LIN {X 0,Y 538.041,Z 253.279,A -85,B 0,C 180,E1 -4113.632,E2 -4113.632} C_VEL
LIN {X 0,Y 538.013,Z 253.279,A -85,B 0,C 180,E1 -4116.121,E2 -4116.121} C_VEL
LIN {X 0,Y 538.043,Z 253.271,A -85,B 0,C 180,E1 -4119.347,E2 -4119.347} C_VEL
LIN {X 0,Y 538.041,Z 253.271,A -85,B 0,C 180,E1 -4122.466,E2 -4122.466} C_VEL
LIN {X 0,Y 538.068,Z 253.272,A -85,B 0,C 180,E1 -4125.629,E2 -4125.629} C_VEL
LIN {X 0,Y 538.081,Z 253.263,A -85,B 0,C 180,E1 -4128.7,E2 -4128.7} C_VEL
LIN {X 0,Y 538.085,Z 253.27,A -85,B 0,C 180,E1 -4131.737,E2 -4131.737} C_VEL
LIN {X 0,Y 538.121,Z 253.267,A -85,B 0,C 180,E1 -4134,E2 -4134} C_VEL
LIN {X 0,Y 538.128,Z 253.259,A -85,B 0,C 180,E1 -4137.003,E2 -4137.003} C_VEL
LIN {X 0,Y 538.174,Z 253.26,A -85,B 0,C 180,E1 -4139.998,E2 -4139.998} C_VEL
LIN {X 0,Y 538.13,Z 253.259,A -85,B 0,C 180,E1 -4142.992,E2 -4142.992} C_VEL
LIN {X 0,Y 538.108,Z 253.267,A -85,B 0,C 180,E1 -4145.995,E2 -4145.995} C_VEL
LIN {X 0,Y 538.055,Z 253.269,A -85,B 0,C 180,E1 -4149.015,E2 -4149.015} C_VEL
LIN {X 0,Y 538.078,Z 253.272,A -85,B 0,C 180,E1 -4152.06,E2 -4152.06} C_VEL
LIN {X 0,Y 538.038,Z 253.27,A -85,B 0,C 180,E1 -4155.141,E2 -4155.141} C_VEL
LIN {X 0,Y 538.017,Z 253.283,A -85,B 0,C 180,E1 -4158.267,E2 -4158.267} C_VEL
LIN {X 0,Y 538.028,Z 253.277,A -85,B 0,C 180,E1 -4160.648,E2 -4160.648} C_VEL
LIN {X 0,Y 537.991,Z 253.279,A -85,B 0,C 180,E1 -4163.885,E2 -4163.885} C_VEL
LIN {X 0,Y 538.029,Z 253.281,A -85,B 0,C 180,E1 -4166.364,E2 -4166.364} C_VEL
LIN {X 0,Y 538.018,Z 253.277,A -85,B 0,C 180,E1 -4168.931,E2 -4168.931} C_VEL
LIN {X 0,Y 537.997,Z 253.277,A -85,B 0,C 180,E1 -4171.885,E2 -4171.885} C_VEL
LIN {X 0,Y 538.008,Z 253.281,A -85,B 0,C 180,E1 -4174.617,E2 -4174.617} C_VEL
LIN {X 0,Y 537.987,Z 253.28,A -85,B 0,C 180,E1 -4177.167,E2 -4177.167} C_VEL
LIN {X 0,Y 538.01,Z 253.276,A -85,B 0,C 180,E1 -4180.241,E2 -4180.241} C_VEL
LIN {X 0,Y 537.37,Z 253.361,A -85,B 0,C 180,E1 -4180.866,E2 -4180.866} C_VEL
LIN {X 0,Y 534.518,Z 253.716,A -85,B 0,C 180,E1 -4181.881,E2 -4181.881} C_VEL
LIN {X 0,Y 532.084,Z 254.023,A -85,B 0,C 180,E1 -4182.698,E2 -4182.698} C_VEL
LIN {X 0,Y 531.029,Z 254.146,A -85,B 0,C 180,E1 -4183.329,E2 -4183.329} C_VEL
LIN {X 0,Y 530.939,Z 254.156,A -85,B 0,C 180,E1 -4183.543,E2 -4183.543} C_VEL
LIN {X 0,Y 530.94,Z 254.163,A -85,B 0,C 180,E1 -4186.503,E2 -4186.503} C_VEL
LIN {X 0,Y 530.982,Z 254.152,A -85,B 0,C 180,E1 -4189.567,E2 -4189.567} C_VEL
LIN {X 0,Y 530.948,Z 254.163,A -85,B 0,C 180,E1 -4192.573,E2 -4192.573} C_VEL
LIN {X 0,Y 530.982,Z 254.156,A -85,B 0,C 180,E1 -4195.31,E2 -4195.31} C_VEL
LIN {X 0,Y 530.884,Z 254.202,A -85,B 0,C 180,E1 -4196.612,E2 -4196.612} C_VEL
LIN {X 0,Y 530.789,Z 266.896,A -85,B 0,C 180,E1 -4199.38,E2 -4199.38} C_VEL
LIN {X 0,Y 530.787,Z 275.719,A -85,B 0,C 180,E1 -4201.314,E2 -4201.314} C_VEL
LIN {X 0,Y 531.967,Z 284.168,A -85,B 0,C 180,E1 -4201.455,E2 -4201.455} C_VEL
LIN {X 0,Y 531.685,Z 351.425,A -85,B 0,C 180,E1 -4202.382,E2 -4202.382} C_VEL
LIN {X 0,Y 531.589,Z 361.171,A -85,B 0,C 180,E1 -4202.624,E2 -4202.624} C_VEL
LIN {X 0,Y 531.484,Z 372.98,A -85,B 0,C 180,E1 -4203.07,E2 -4203.07} C_VEL
LIN {X 0,Y 531.329,Z 382.663,A -85,B 0,C 180,E1 -4203.592,E2 -4203.592} C_VEL
LIN {X 0,Y 531.152,Z 391.309,A -85,B 0,C 180,E1 -4204.186,E2 -4204.186} C_VEL
LIN {X 0,Y 530.989,Z 398.99,A -85,B 0,C 180,E1 -4204.837,E2 -4204.837} C_VEL
LIN {X 0,Y 530.851,Z 406.002,A -85,B 0,C 180,E1 -4205.561,E2 -4205.561} C_VEL
LIN {X 0,Y 530.738,Z 412.812,A -85,B 0,C 180,E1 -4206.42,E2 -4206.42} C_VEL
LIN {X 0,Y 530.635,Z 419.151,A -85,B 0,C 180,E1 -4207.413,E2 -4207.413} C_VEL
LIN {X 0,Y 530.543,Z 423.279,A -85,B 0,C 180,E1 -4208.228,E2 -4208.228} C_VEL
LIN {X 0,Y 530.505,Z 427.975,A -85,B 0,C 180,E1 -4209.448,E2 -4209.448} C_VEL
LIN {X 0,Y 530.483,Z 430.043,A -85,B 0,C 180,E1 -4210.145,E2 -4210.145} C_VEL
LIN {X 0,Y 530.384,Z 432.54,A -85,B 0,C 180,E1 -4211.457,E2 -4211.457} C_VEL
LIN {X 0,Y 530.398,Z 433.506,A -85,B 0,C 180,E1 -4212.545,E2 -4212.545} C_VEL
LIN {X 0,Y 530.42,Z 433.688,A -85,B 0,C 180,E1 -4213.053,E2 -4213.053} C_VEL
LIN {X 0,Y 530.396,Z 433.379,A -85,B 0,C 180,E1 -4213.844,E2 -4213.844} C_VEL
LIN {X 0,Y 530.412,Z 432.535,A -85,B 0,C 180,E1 -4214.633,E2 -4214.633} C_VEL
LIN {X 0,Y 530.456,Z 431.175,A -85,B 0,C 180,E1 -4215.42,E2 -4215.42} C_VEL
LIN {X 0,Y 530.509,Z 428.107,A -85,B 0,C 180,E1 -4216.595,E2 -4216.595} C_VEL
LIN {X 0,Y 530.556,Z 423.719,A -85,B 0,C 180,E1 -4217.764,E2 -4217.764} C_VEL
LIN {X 0,Y 530.654,Z 419.171,A -85,B 0,C 180,E1 -4218.671,E2 -4218.671} C_VEL
LIN {X 0,Y 530.728,Z 412.559,A -85,B 0,C 180,E1 -4219.702,E2 -4219.702} C_VEL
LIN {X 0,Y 530.856,Z 406.455,A -85,B 0,C 180,E1 -4220.475,E2 -4220.475} C_VEL
LIN {X 0,Y 531.014,Z 399.031,A -85,B 0,C 180,E1 -4221.246,E2 -4221.246} C_VEL
LIN {X 0,Y 531.138,Z 391.103,A -85,B 0,C 180,E1 -4221.918,E2 -4221.918} C_VEL
LIN {X 0,Y 531.308,Z 381.979,A -85,B 0,C 180,E1 -4222.54,E2 -4222.54} C_VEL
LIN {X 0,Y 531.46,Z 371.213,A -85,B 0,C 180,E1 -4223.097,E2 -4223.097} C_VEL
LIN {X 0,Y 531.575,Z 360.799,A -85,B 0,C 180,E1 -4223.476,E2 -4223.476} C_VEL
LIN {X 0,Y 531.7,Z 350.946,A -85,B 0,C 180,E1 -4223.716,E2 -4223.716} C_VEL
LIN {X 0,Y 531.779,Z 281.945,A -85,B 0,C 180,E1 -4224.668,E2 -4224.668} C_VEL
LIN {X 0,Y 530.812,Z 275.687,A -85,B 0,C 180,E1 -4224.778,E2 -4224.778} C_VEL
LIN {X 0,Y 530.914,Z 261.115,A -85,B 0,C 180,E1 -4228.104,E2 -4228.104} C_VEL
LIN {X 0,Y 530.937,Z 254.161,A -85,B 0,C 180,E1 -4229.716,E2 -4229.716} C_VEL
LIN {X 0,Y 531.118,Z 254.139,A -85,B 0,C 180,E1 -4230.758,E2 -4230.758} C_VEL
LIN {X 0,Y 531.072,Z 254.145,A -85,B 0,C 180,E1 -4233.034,E2 -4233.034} C_VEL
LIN {X 0,Y 531.04,Z 254.144,A -85,B 0,C 180,E1 -4236.078,E2 -4236.078} C_VEL
LIN {X 0,Y 530.988,Z 254.157,A -85,B 0,C 180,E1 -4239.139,E2 -4239.139} C_VEL
LIN {X 0,Y 531.021,Z 254.15,A -85,B 0,C 180,E1 -4241.677,E2 -4241.677} C_VEL
LIN {X 0,Y 530.991,Z 254.153,A -85,B 0,C 180,E1 -4244.956,E2 -4244.956} C_VEL
LIN {X 0,Y 530.979,Z 254.155,A -85,B 0,C 180,E1 -4247.724,E2 -4247.724} C_VEL
LIN {X 0,Y 530.988,Z 254.15,A -85,B 0,C 180,E1 -4250.129,E2 -4250.129} C_VEL
LIN {X 0,Y 530.907,Z 254.16,A -85,B 0,C 180,E1 -4252.575,E2 -4252.575} C_VEL
LIN {X 0,Y 530.925,Z 254.161,A -85,B 0,C 180,E1 -4255.062,E2 -4255.062} C_VEL
LIN {X 0,Y 530.937,Z 254.164,A -85,B 0,C 180,E1 -4257.6,E2 -4257.6} C_VEL
LIN {X 0,Y 530.926,Z 254.158,A -85,B 0,C 180,E1 -4260.2,E2 -4260.2} C_VEL
LIN {X 0,Y 530.936,Z 254.157,A -85,B 0,C 180,E1 -4262.869,E2 -4262.869} C_VEL
LIN {X 0,Y 530.919,Z 254.167,A -85,B 0,C 180,E1 -4265.623,E2 -4265.623} C_VEL
LIN {X 0,Y 530.933,Z 254.157,A -85,B 0,C 180,E1 -4268.656,E2 -4268.656} C_VEL
LIN {X 0,Y 530.952,Z 254.161,A -85,B 0,C 180,E1 -4271.44,E2 -4271.44} C_VEL
LIN {X 0,Y 530.949,Z 254.155,A -85,B 0,C 180,E1 -4274.551,E2 -4274.551} C_VEL
LIN {X 0,Y 530.96,Z 254.16,A -85,B 0,C 180,E1 -4277.837,E2 -4277.837} C_VEL
LIN {X 0,Y 530.963,Z 254.153,A -85,B 0,C 180,E1 -4280.559,E2 -4280.559} C_VEL
LIN {X 0,Y 530.934,Z 254.162,A -85,B 0,C 180,E1 -4283.444,E2 -4283.444} C_VEL
LIN {X 0,Y 530.939,Z 254.158,A -85,B 0,C 180,E1 -4286.228,E2 -4286.228} C_VEL
LIN {X 0,Y 530.96,Z 254.158,A -85,B 0,C 180,E1 -4289.358,E2 -4289.358} C_VEL
LIN {X 0,Y 530.951,Z 254.161,A -85,B 0,C 180,E1 -4291.546,E2 -4291.546} C_VEL
LIN {X 0,Y 530.963,Z 254.157,A -85,B 0,C 180,E1 -4294.168,E2 -4294.168} C_VEL
LIN {X 0,Y 530.943,Z 254.156,A -85,B 0,C 180,E1 -4296.606,E2 -4296.606} C_VEL
LIN {X 0,Y 530.99,Z 254.151,A -85,B 0,C 180,E1 -4299.065,E2 -4299.065} C_VEL
LIN {X 0,Y 530.964,Z 254.158,A -85,B 0,C 180,E1 -4301.481,E2 -4301.481} C_VEL
LIN {X 0,Y 530.961,Z 254.324,A -85,B 0,C 180,E1 -4303.321,E2 -4303.321} C_VEL
LIN {X 0,Y 530.917,Z 265.036,A -85,B 0,C 180,E1 -4305.828,E2 -4305.828} C_VEL
LIN {X 0,Y 530.785,Z 275.645,A -85,B 0,C 180,E1 -4308.323,E2 -4308.323} C_VEL
LIN {X 0,Y 531.892,Z 283.251,A -85,B 0,C 180,E1 -4308.465,E2 -4308.465} C_VEL
LIN {X 0,Y 531.64,Z 352.125,A -85,B 0,C 180,E1 -4309.434,E2 -4309.434} C_VEL
LIN {X 0,Y 531.525,Z 363.522,A -85,B 0,C 180,E1 -4309.744,E2 -4309.744} C_VEL
LIN {X 0,Y 531.334,Z 374.684,A -85,B 0,C 180,E1 -4310.198,E2 -4310.198} C_VEL
LIN {X 0,Y 531.216,Z 384.815,A -85,B 0,C 180,E1 -4310.772,E2 -4310.772} C_VEL
LIN {X 0,Y 531.091,Z 393.972,A -85,B 0,C 180,E1 -4311.441,E2 -4311.441} C_VEL
LIN {X 0,Y 530.918,Z 402.344,A -85,B 0,C 180,E1 -4312.205,E2 -4312.205} C_VEL
LIN {X 0,Y 530.758,Z 410.574,A -85,B 0,C 180,E1 -4313.158,E2 -4313.158} C_VEL
LIN {X 0,Y 530.717,Z 417.097,A -85,B 0,C 180,E1 -4314.112,E2 -4314.112} C_VEL
LIN {X 0,Y 530.581,Z 422.263,A -85,B 0,C 180,E1 -4315.063,E2 -4315.063} C_VEL
LIN {X 0,Y 530.56,Z 425.573,A -85,B 0,C 180,E1 -4315.825,E2 -4315.825} C_VEL
LIN {X 0,Y 530.527,Z 429.412,A -85,B 0,C 180,E1 -4316.965,E2 -4316.965} C_VEL
LIN {X 0,Y 530.412,Z 431.261,A -85,B 0,C 180,E1 -4317.724,E2 -4317.724} C_VEL
LIN {X 0,Y 530.363,Z 432.569,A -85,B 0,C 180,E1 -4318.484,E2 -4318.484} C_VEL
LIN {X 0,Y 530.355,Z 433.359,A -85,B 0,C 180,E1 -4319.243,E2 -4319.243} C_VEL
LIN {X 0,Y 530.357,Z 433.615,A -85,B 0,C 180,E1 -4320.002,E2 -4320.002} C_VEL
LIN {X 0,Y 530.357,Z 433.432,A -85,B 0,C 180,E1 -4320.762,E2 -4320.762} C_VEL
LIN {X 0,Y 530.363,Z 432.692,A -85,B 0,C 180,E1 -4321.521,E2 -4321.521} C_VEL
LIN {X 0,Y 530.414,Z 431.453,A -85,B 0,C 180,E1 -4322.28,E2 -4322.28} C_VEL
LIN {X 0,Y 530.549,Z 428.597,A -85,B 0,C 180,E1 -4323.42,E2 -4323.42} C_VEL
LIN {X 0,Y 530.604,Z 424.486,A -85,B 0,C 180,E1 -4324.56,E2 -4324.56} C_VEL
LIN {X 0,Y 530.659,Z 418.8,A -85,B 0,C 180,E1 -4325.703,E2 -4325.703} C_VEL
LIN {X 0,Y 530.729,Z 412.348,A -85,B 0,C 180,E1 -4326.702,E2 -4326.702} C_VEL
LIN {X 0,Y 530.87,Z 404.997,A -85,B 0,C 180,E1 -4327.61,E2 -4327.61} C_VEL
LIN {X 0,Y 531.037,Z 396.186,A -85,B 0,C 180,E1 -4328.469,E2 -4328.469} C_VEL
LIN {X 0,Y 531.245,Z 387.509,A -85,B 0,C 180,E1 -4329.137,E2 -4329.137} C_VEL
LIN {X 0,Y 531.351,Z 378.086,A -85,B 0,C 180,E1 -4329.711,E2 -4329.711} C_VEL
LIN {X 0,Y 531.489,Z 367.857,A -85,B 0,C 180,E1 -4330.189,E2 -4330.189} C_VEL
LIN {X 0,Y 531.58,Z 356.589,A -85,B 0,C 180,E1 -4330.548,E2 -4330.548} C_VEL
LIN {X 0,Y 531.737,Z 343.655,A -85,B 0,C 180,E1 -4330.786,E2 -4330.786} C_VEL
LIN {X 0,Y 531.751,Z 281.777,A -85,B 0,C 180,E1 -4331.649,E2 -4331.649} C_VEL
LIN {X 0,Y 530.789,Z 275.755,A -85,B 0,C 180,E1 -4331.767,E2 -4331.767} C_VEL
LIN {X 0,Y 530.888,Z 265.704,A -85,B 0,C 180,E1 -4334.178,E2 -4334.178} C_VEL
LIN {X 0,Y 531.002,Z 254.155,A -85,B 0,C 180,E1 -4336.782,E2 -4336.782} C_VEL
LIN {X 0,Y 531.033,Z 254.155,A -85,B 0,C 180,E1 -4340.129,E2 -4340.129} C_VEL
LIN {X 0,Y 530.951,Z 254.161,A -85,B 0,C 180,E1 -4342.575,E2 -4342.575} C_VEL
LIN {X 0,Y 530.959,Z 254.156,A -85,B 0,C 180,E1 -4345.062,E2 -4345.062} C_VEL
LIN {X 0,Y 530.973,Z 254.154,A -85,B 0,C 180,E1 -4347.599,E2 -4347.599} C_VEL
LIN {X 0,Y 530.961,Z 254.161,A -85,B 0,C 180,E1 -4350.199,E2 -4350.199} C_VEL
LIN {X 0,Y 530.975,Z 254.156,A -85,B 0,C 180,E1 -4352.868,E2 -4352.868} C_VEL
LIN {X 0,Y 530.956,Z 254.155,A -85,B 0,C 180,E1 -4355.621,E2 -4355.621} C_VEL
LIN {X 0,Y 530.971,Z 254.16,A -85,B 0,C 180,E1 -4358.654,E2 -4358.654} C_VEL
LIN {X 0,Y 530.987,Z 254.151,A -85,B 0,C 180,E1 -4361.438,E2 -4361.438} C_VEL
LIN {X 0,Y 530.98,Z 254.159,A -85,B 0,C 180,E1 -4364.549,E2 -4364.549} C_VEL
LIN {X 0,Y 530.976,Z 254.152,A -85,B 0,C 180,E1 -4367.836,E2 -4367.836} C_VEL
LIN {X 0,Y 530.99,Z 254.158,A -85,B 0,C 180,E1 -4370.557,E2 -4370.557} C_VEL
LIN {X 0,Y 530.957,Z 254.153,A -85,B 0,C 180,E1 -4373.441,E2 -4373.441} C_VEL
LIN {X 0,Y 530.961,Z 254.156,A -85,B 0,C 180,E1 -4376.225,E2 -4376.225} C_VEL
LIN {X 0,Y 530.96,Z 254.161,A -85,B 0,C 180,E1 -4378.921,E2 -4378.921} C_VEL
LIN {X 0,Y 530.978,Z 254.153,A -85,B 0,C 180,E1 -4381.543,E2 -4381.543} C_VEL
LIN {X 0,Y 531.018,Z 254.149,A -85,B 0,C 180,E1 -4384.156,E2 -4384.156} C_VEL
LIN {X 0,Y 531.044,Z 254.342,A -85,B 0,C 180,E1 -4386.814,E2 -4386.814} C_VEL
LIN {X 0,Y 531.791,Z 259.167,A -85,B 0,C 180,E1 -4387.685,E2 -4387.685} C_VEL
LIN {X 0,Y 531.629,Z 273.173,A -85,B 0,C 180,E1 -4390.098,E2 -4390.098} C_VEL
LIN {X 0,Y 531.34,Z 289.579,A -85,B 0,C 180,E1 -4392.884,E2 -4392.884} C_VEL
LIN {X 0,Y 531.07,Z 308.295,A -85,B 0,C 180,E1 -4396.024,E2 -4396.024} C_VEL
LIN {X 0,Y 530.887,Z 321.55,A -85,B 0,C 180,E1 -4398.231,E2 -4398.231} C_VEL
LIN {X 0,Y 531.888,Z 330.701,A -85,B 0,C 180,E1 -4398.389,E2 -4398.389} C_VEL
LIN {X 0,Y 531.659,Z 399.476,A -85,B 0,C 180,E1 -4399.335,E2 -4399.335} C_VEL
LIN {X 0,Y 531.516,Z 409.998,A -85,B 0,C 180,E1 -4399.597,E2 -4399.597} C_VEL
LIN {X 0,Y 531.364,Z 420.758,A -85,B 0,C 180,E1 -4400.003,E2 -4400.003} C_VEL
LIN {X 0,Y 531.221,Z 431.422,A -85,B 0,C 180,E1 -4400.577,E2 -4400.577} C_VEL
LIN {X 0,Y 531.118,Z 439.774,A -85,B 0,C 180,E1 -4401.151,E2 -4401.151} C_VEL
LIN {X 0,Y 530.931,Z 447.675,A -85,B 0,C 180,E1 -4401.819,E2 -4401.819} C_VEL
LIN {X 0,Y 530.786,Z 455.064,A -85,B 0,C 180,E1 -4402.582,E2 -4402.582} C_VEL
LIN {X 0,Y 530.669,Z 462.835,A -85,B 0,C 180,E1 -4403.575,E2 -4403.575} C_VEL
LIN {X 0,Y 530.542,Z 469.414,A -85,B 0,C 180,E1 -4404.679,E2 -4404.679} C_VEL
LIN {X 0,Y 530.544,Z 474.617,A -85,B 0,C 180,E1 -4405.822,E2 -4405.822} C_VEL
LIN {X 0,Y 530.47,Z 478.434,A -85,B 0,C 180,E1 -4406.962,E2 -4406.962} C_VEL
LIN {X 0,Y 530.413,Z 480.189,A -85,B 0,C 180,E1 -4407.722,E2 -4407.722} C_VEL
LIN {X 0,Y 530.36,Z 481.446,A -85,B 0,C 180,E1 -4408.481,E2 -4408.481} C_VEL
LIN {X 0,Y 530.347,Z 482.23,A -85,B 0,C 180,E1 -4409.241,E2 -4409.241} C_VEL
LIN {X 0,Y 530.349,Z 482.526,A -85,B 0,C 180,E1 -4410,E2 -4410} C_VEL
LIN {X 0,Y 530.347,Z 482.228,A -85,B 0,C 180,E1 -4410.759,E2 -4410.759} C_VEL
LIN {X 0,Y 530.36,Z 481.444,A -85,B 0,C 180,E1 -4411.519,E2 -4411.519} C_VEL
LIN {X 0,Y 530.413,Z 480.185,A -85,B 0,C 180,E1 -4412.278,E2 -4412.278} C_VEL
LIN {X 0,Y 530.494,Z 477.269,A -85,B 0,C 180,E1 -4413.418,E2 -4413.418} C_VEL
LIN {X 0,Y 530.544,Z 474.61,A -85,B 0,C 180,E1 -4414.178,E2 -4414.178} C_VEL
LIN {X 0,Y 530.542,Z 469.402,A -85,B 0,C 180,E1 -4415.32,E2 -4415.32} C_VEL
LIN {X 0,Y 530.673,Z 462.787,A -85,B 0,C 180,E1 -4416.429,E2 -4416.429} C_VEL
LIN {X 0,Y 530.786,Z 455.052,A -85,B 0,C 180,E1 -4417.417,E2 -4417.417} C_VEL
LIN {X 0,Y 530.929,Z 447.664,A -85,B 0,C 180,E1 -4418.181,E2 -4418.181} C_VEL
LIN {X 0,Y 531.097,Z 439.756,A -85,B 0,C 180,E1 -4418.849,E2 -4418.849} C_VEL
LIN {X 0,Y 531.221,Z 431.401,A -85,B 0,C 180,E1 -4419.423,E2 -4419.423} C_VEL
LIN {X 0,Y 531.364,Z 420.737,A -85,B 0,C 180,E1 -4419.997,E2 -4419.997} C_VEL
LIN {X 0,Y 531.525,Z 409.145,A -85,B 0,C 180,E1 -4420.427,E2 -4420.427} C_VEL
LIN {X 0,Y 531.652,Z 399.452,A -85,B 0,C 180,E1 -4420.665,E2 -4420.665} C_VEL
LIN {X 0,Y 531.882,Z 330.638,A -85,B 0,C 180,E1 -4421.612,E2 -4421.612} C_VEL
LIN {X 0,Y 530.891,Z 321.475,A -85,B 0,C 180,E1 -4421.77,E2 -4421.77} C_VEL
LIN {X 0,Y 531.107,Z 302.114,A -85,B 0,C 180,E1 -4424.985,E2 -4424.985} C_VEL
LIN {X 0,Y 531.411,Z 283.707,A -85,B 0,C 180,E1 -4428.067,E2 -4428.067} C_VEL
LIN {X 0,Y 531.701,Z 265.728,A -85,B 0,C 180,E1 -4431.112,E2 -4431.112} C_VEL
LIN {X 0,Y 531.732,Z 258.797,A -85,B 0,C 180,E1 -4432.3,E2 -4432.3} C_VEL
LIN {X 0,Y 531.015,Z 254.156,A -85,B 0,C 180,E1 -4433.136,E2 -4433.136} C_VEL
LIN {X 0,Y 531.016,Z 254.149,A -85,B 0,C 180,E1 -4435.897,E2 -4435.897} C_VEL
LIN {X 0,Y 530.976,Z 254.153,A -85,B 0,C 180,E1 -4438.457,E2 -4438.457} C_VEL
LIN {X 0,Y 530.958,Z 254.16,A -85,B 0,C 180,E1 -4441.079,E2 -4441.079} C_VEL
LIN {X 0,Y 530.96,Z 254.158,A -85,B 0,C 180,E1 -4443.775,E2 -4443.775} C_VEL
LIN {X 0,Y 530.959,Z 254.152,A -85,B 0,C 180,E1 -4446.558,E2 -4446.558} C_VEL
LIN {X 0,Y 530.989,Z 254.159,A -85,B 0,C 180,E1 -4449.443,E2 -4449.443} C_VEL
LIN {X 0,Y 530.979,Z 254.151,A -85,B 0,C 180,E1 -4452.456,E2 -4452.456} C_VEL
LIN {X 0,Y 530.981,Z 254.159,A -85,B 0,C 180,E1 -4455.622,E2 -4455.622} C_VEL
LIN {X 0,Y 530.999,Z 254.148,A -85,B 0,C 180,E1 -4458.563,E2 -4458.563} C_VEL
LIN {X 0,Y 530.961,Z 254.16,A -85,B 0,C 180,E1 -4461.528,E2 -4461.528} C_VEL
LIN {X 0,Y 530.959,Z 254.152,A -85,B 0,C 180,E1 -4464.379,E2 -4464.379} C_VEL
LIN {X 0,Y 530.972,Z 254.154,A -85,B 0,C 180,E1 -4467.132,E2 -4467.132} C_VEL
LIN {X 0,Y 530.96,Z 254.161,A -85,B 0,C 180,E1 -4469.801,E2 -4469.801} C_VEL
LIN {X 0,Y 530.979,Z 254.151,A -85,B 0,C 180,E1 -4472.475,E2 -4472.475} C_VEL
LIN {X 0,Y 530.994,Z 254.149,A -85,B 0,C 180,E1 -4474.94,E2 -4474.94} C_VEL
LIN {X 0,Y 530.977,Z 254.152,A -85,B 0,C 180,E1 -4478.245,E2 -4478.245} C_VEL
LIN {X 0,Y 530.988,Z 254.15,A -85,B 0,C 180,E1 -4480.675,E2 -4480.675} C_VEL
LIN {X 0,Y 530.974,Z 254.15,A -85,B 0,C 180,E1 -4483.069,E2 -4483.069} C_VEL
LIN {X 0,Y 531.024,Z 254.146,A -85,B 0,C 180,E1 -4485.434,E2 -4485.434} C_VEL
LIN {X 0,Y 531.039,Z 254.141,A -85,B 0,C 180,E1 -4488.548,E2 -4488.548} C_VEL
LIN {X 0,Y 531.054,Z 254.144,A -85,B 0,C 180,E1 -4491.627,E2 -4491.627} C_VEL
LIN {X 0,Y 531.119,Z 254.131,A -85,B 0,C 180,E1 -4494.683,E2 -4494.683} C_VEL
LIN {X 0,Y 531.14,Z 254.134,A -85,B 0,C 180,E1 -4497.723,E2 -4497.723} C_VEL
LIN {X 0,Y 531.147,Z 254.129,A -85,B 0,C 180,E1 -4500.756,E2 -4500.756} C_VEL
LIN {X 0,Y 531.098,Z 254.135,A -85,B 0,C 180,E1 -4503.032,E2 -4503.032} C_VEL
LIN {X 0,Y 531.064,Z 254.145,A -85,B 0,C 180,E1 -4506.075,E2 -4506.075} C_VEL
LIN {X 0,Y 531.015,Z 254.145,A -85,B 0,C 180,E1 -4509.136,E2 -4509.136} C_VEL
LIN {X 0,Y 531.035,Z 254.152,A -85,B 0,C 180,E1 -4512.222,E2 -4512.222} C_VEL
LIN {X 0,Y 530.988,Z 254.148,A -85,B 0,C 180,E1 -4515.347,E2 -4515.347} C_VEL
LIN {X 0,Y 530.977,Z 254.157,A -85,B 0,C 180,E1 -4518.518,E2 -4518.518} C_VEL
LIN {X 0,Y 530.989,Z 254.151,A -85,B 0,C 180,E1 -4520.935,E2 -4520.935} C_VEL
LIN {X 0,Y 530.959,Z 254.16,A -85,B 0,C 180,E1 -4524.222,E2 -4524.222} C_VEL
LIN {X 0,Y 530.993,Z 254.154,A -85,B 0,C 180,E1 -4526.741,E2 -4526.741} C_VEL
LIN {X 0,Y 530.968,Z 254.153,A -85,B 0,C 180,E1 -4529.319,E2 -4529.319} C_VEL
LIN {X 0,Y 530.953,Z 254.157,A -85,B 0,C 180,E1 -4532.098,E2 -4532.098} C_VEL
LIN {X 0,Y 530.965,Z 254.155,A -85,B 0,C 180,E1 -4534.85,E2 -4534.85} C_VEL
LIN {X 0,Y 530.946,Z 254.155,A -85,B 0,C 180,E1 -4537.505,E2 -4537.505} C_VEL
LIN {X 0,Y 530.978,Z 254.157,A -85,B 0,C 180,E1 -4540.428,E2 -4540.428} C_VEL
LIN {X 0,Y 530.942,Z 254.156,A -85,B 0,C 180,E1 -4543.492,E2 -4543.492} C_VEL
LIN {X 0,Y 530.939,Z 254.156,A -85,B 0,C 180,E1 -4543.543,E2 -4543.543} C_VEL
LIN {X 0,Y 530.264,Z 254.243,A -85,B 0,C 180,E1 -4544.176,E2 -4544.176} C_VEL
LIN {X 0,Y 527.417,Z 254.604,A -85,B 0,C 180,E1 -4545.205,E2 -4545.205} C_VEL
LIN {X 0,Y 525.015,Z 254.906,A -85,B 0,C 180,E1 -4546.034,E2 -4546.034} C_VEL
LIN {X 0,Y 523.983,Z 255.032,A -85,B 0,C 180,E1 -4546.673,E2 -4546.673} C_VEL
LIN {X 0,Y 523.898,Z 255.04,A -85,B 0,C 180,E1 -4546.89,E2 -4546.89} C_VEL
LIN {X 0,Y 523.94,Z 255.029,A -85,B 0,C 180,E1 -4549.864,E2 -4549.864} C_VEL
LIN {X 0,Y 523.888,Z 255.044,A -85,B 0,C 180,E1 -4552.866,E2 -4552.866} C_VEL
LIN {X 0,Y 523.938,Z 255.032,A -85,B 0,C 180,E1 -4555.71,E2 -4555.71} C_VEL
LIN {X 0,Y 523.813,Z 255.215,A -85,B 0,C 180,E1 -4556.626,E2 -4556.626} C_VEL
LIN {X 0,Y 523.765,Z 268.683,A -85,B 0,C 180,E1 -4559.567,E2 -4559.567} C_VEL
LIN {X 0,Y 523.74,Z 275.82,A -85,B 0,C 180,E1 -4561.15,E2 -4561.15} C_VEL
LIN {X 0,Y 525.046,Z 284.56,A -85,B 0,C 180,E1 -4561.301,E2 -4561.301} C_VEL
LIN {X 0,Y 524.723,Z 351.234,A -85,B 0,C 180,E1 -4562.23,E2 -4562.23} C_VEL
LIN {X 0,Y 524.627,Z 360.645,A -85,B 0,C 180,E1 -4562.459,E2 -4562.459} C_VEL
LIN {X 0,Y 524.523,Z 369.883,A -85,B 0,C 180,E1 -4562.791,E2 -4562.791} C_VEL
LIN {X 0,Y 524.36,Z 380.685,A -85,B 0,C 180,E1 -4563.321,E2 -4563.321} C_VEL
LIN {X 0,Y 524.209,Z 390.837,A -85,B 0,C 180,E1 -4564.005,E2 -4564.005} C_VEL
LIN {X 0,Y 523.978,Z 398.921,A -85,B 0,C 180,E1 -4564.689,E2 -4564.689} C_VEL
LIN {X 0,Y 523.825,Z 406.001,A -85,B 0,C 180,E1 -4565.423,E2 -4565.423} C_VEL
LIN {X 0,Y 523.708,Z 412.619,A -85,B 0,C 180,E1 -4566.26,E2 -4566.26} C_VEL
LIN {X 0,Y 523.59,Z 419.266,A -85,B 0,C 180,E1 -4567.301,E2 -4567.301} C_VEL
LIN {X 0,Y 523.471,Z 424.36,A -85,B 0,C 180,E1 -4568.333,E2 -4568.333} C_VEL
LIN {X 0,Y 523.439,Z 427.555,A -85,B 0,C 180,E1 -4569.157,E2 -4569.157} C_VEL
LIN {X 0,Y 523.36,Z 430.981,A -85,B 0,C 180,E1 -4570.384,E2 -4570.384} C_VEL
LIN {X 0,Y 523.3,Z 432.571,A -85,B 0,C 180,E1 -4571.197,E2 -4571.197} C_VEL
LIN {X 0,Y 523.31,Z 433.566,A -85,B 0,C 180,E1 -4572.008,E2 -4572.008} C_VEL
LIN {X 0,Y 523.323,Z 433.946,A -85,B 0,C 180,E1 -4572.816,E2 -4572.816} C_VEL
LIN {X 0,Y 523.301,Z 433.803,A -85,B 0,C 180,E1 -4573.619,E2 -4573.619} C_VEL
LIN {X 0,Y 523.329,Z 433.151,A -85,B 0,C 180,E1 -4574.42,E2 -4574.42} C_VEL
LIN {X 0,Y 523.342,Z 431.99,A -85,B 0,C 180,E1 -4575.218,E2 -4575.218} C_VEL
LIN {X 0,Y 523.41,Z 430.284,A -85,B 0,C 180,E1 -4576.014,E2 -4576.014} C_VEL
LIN {X 0,Y 523.43,Z 426.518,A -85,B 0,C 180,E1 -4577.2,E2 -4577.2} C_VEL
LIN {X 0,Y 523.521,Z 421.341,A -85,B 0,C 180,E1 -4578.383,E2 -4578.383} C_VEL
LIN {X 0,Y 523.666,Z 415.766,A -85,B 0,C 180,E1 -4579.366,E2 -4579.366} C_VEL
LIN {X 0,Y 523.768,Z 408.78,A -85,B 0,C 180,E1 -4580.344,E2 -4580.344} C_VEL
LIN {X 0,Y 523.936,Z 400.743,A -85,B 0,C 180,E1 -4581.224,E2 -4581.224} C_VEL
LIN {X 0,Y 524.119,Z 393.072,A -85,B 0,C 180,E1 -4581.906,E2 -4581.906} C_VEL
LIN {X 0,Y 524.273,Z 385.49,A -85,B 0,C 180,E1 -4582.46,E2 -4582.46} C_VEL
LIN {X 0,Y 524.375,Z 378.301,A -85,B 0,C 180,E1 -4582.893,E2 -4582.893} C_VEL
LIN {X 0,Y 524.502,Z 369.433,A -85,B 0,C 180,E1 -4583.315,E2 -4583.315} C_VEL
LIN {X 0,Y 524.618,Z 360.593,A -85,B 0,C 180,E1 -4583.631,E2 -4583.631} C_VEL
LIN {X 0,Y 524.728,Z 351.763,A -85,B 0,C 180,E1 -4583.849,E2 -4583.849} C_VEL
LIN {X 0,Y 524.873,Z 282.897,A -85,B 0,C 180,E1 -4584.815,E2 -4584.815} C_VEL
LIN {X 0,Y 523.778,Z 275.848,A -85,B 0,C 180,E1 -4584.948,E2 -4584.948} C_VEL
LIN {X 0,Y 523.896,Z 260.476,A -85,B 0,C 180,E1 -4588.463,E2 -4588.463} C_VEL
LIN {X 0,Y 523.896,Z 255.038,A -85,B 0,C 180,E1 -4589.712,E2 -4589.712} C_VEL
LIN {X 0,Y 524.088,Z 255.015,A -85,B 0,C 180,E1 -4590.769,E2 -4590.769} C_VEL
LIN {X 0,Y 524.039,Z 255.022,A -85,B 0,C 180,E1 -4593.075,E2 -4593.075} C_VEL
LIN {X 0,Y 524.001,Z 255.021,A -85,B 0,C 180,E1 -4596.16,E2 -4596.16} C_VEL
LIN {X 0,Y 523.961,Z 255.025,A -85,B 0,C 180,E1 -4598.485,E2 -4598.485} C_VEL
LIN {X 0,Y 523.97,Z 255.028,A -85,B 0,C 180,E1 -4601.744,E2 -4601.744} C_VEL
LIN {X 0,Y 523.953,Z 255.031,A -85,B 0,C 180,E1 -4605.053,E2 -4605.053} C_VEL
LIN {X 0,Y 523.926,Z 255.031,A -85,B 0,C 180,E1 -4607.971,E2 -4607.971} C_VEL
LIN {X 0,Y 523.935,Z 255.028,A -85,B 0,C 180,E1 -4610.412,E2 -4610.412} C_VEL
LIN {X 0,Y 523.873,Z 255.038,A -85,B 0,C 180,E1 -4612.896,E2 -4612.896} C_VEL
LIN {X 0,Y 523.874,Z 255.045,A -85,B 0,C 180,E1 -4615.423,E2 -4615.423} C_VEL
LIN {X 0,Y 523.885,Z 255.037,A -85,B 0,C 180,E1 -4618.004,E2 -4618.004} C_VEL
LIN {X 0,Y 523.906,Z 255.033,A -85,B 0,C 180,E1 -4620.856,E2 -4620.856} C_VEL
LIN {X 0,Y 523.928,Z 255.035,A -85,B 0,C 180,E1 -4623.737,E2 -4623.737} C_VEL
LIN {X 0,Y 523.868,Z 255.037,A -85,B 0,C 180,E1 -4626.403,E2 -4626.403} C_VEL
LIN {X 0,Y 523.884,Z 255.037,A -85,B 0,C 180,E1 -4629.088,E2 -4629.088} C_VEL
LIN {X 0,Y 523.913,Z 255.033,A -85,B 0,C 180,E1 -4632.123,E2 -4632.123} C_VEL
LIN {X 0,Y 523.919,Z 255.035,A -85,B 0,C 180,E1 -4635.313,E2 -4635.313} C_VEL
LIN {X 0,Y 523.935,Z 255.029,A -85,B 0,C 180,E1 -4638.693,E2 -4638.693} C_VEL
LIN {X 0,Y 523.895,Z 255.035,A -85,B 0,C 180,E1 -4641.084,E2 -4641.084} C_VEL
LIN {X 0,Y 523.881,Z 255.043,A -85,B 0,C 180,E1 -4643.828,E2 -4643.828} C_VEL
LIN {X 0,Y 523.897,Z 255.034,A -85,B 0,C 180,E1 -4646.637,E2 -4646.637} C_VEL
LIN {X 0,Y 523.941,Z 255.032,A -85,B 0,C 180,E1 -4649.359,E2 -4649.359} C_VEL
LIN {X 0,Y 523.928,Z 255.032,A -85,B 0,C 180,E1 -4652.292,E2 -4652.292} C_VEL
LIN {X 0,Y 523.908,Z 255.037,A -85,B 0,C 180,E1 -4655.431,E2 -4655.431} C_VEL
LIN {X 0,Y 523.929,Z 255.037,A -85,B 0,C 180,E1 -4657.943,E2 -4657.943} C_VEL
LIN {X 0,Y 523.96,Z 255.028,A -85,B 0,C 180,E1 -4660.411,E2 -4660.411} C_VEL
LIN {X 0,Y 523.93,Z 255.119,A -85,B 0,C 180,E1 -4663.291,E2 -4663.291} C_VEL
LIN {X 0,Y 523.833,Z 266.792,A -85,B 0,C 180,E1 -4666.028,E2 -4666.028} C_VEL
LIN {X 0,Y 523.724,Z 275.885,A -85,B 0,C 180,E1 -4668.167,E2 -4668.167} C_VEL
LIN {X 0,Y 524.939,Z 285.179,A -85,B 0,C 180,E1 -4668.337,E2 -4668.337} C_VEL
LIN {X 0,Y 524.674,Z 351.745,A -85,B 0,C 180,E1 -4669.292,E2 -4669.292} C_VEL
LIN {X 0,Y 524.546,Z 362.616,A -85,B 0,C 180,E1 -4669.582,E2 -4669.582} C_VEL
LIN {X 0,Y 524.389,Z 372.506,A -85,B 0,C 180,E1 -4669.969,E2 -4669.969} C_VEL
LIN {X 0,Y 524.263,Z 383.419,A -85,B 0,C 180,E1 -4670.551,E2 -4670.551} C_VEL
LIN {X 0,Y 524.119,Z 392.899,A -85,B 0,C 180,E1 -4671.229,E2 -4671.229} C_VEL
LIN {X 0,Y 523.935,Z 400.533,A -85,B 0,C 180,E1 -4671.906,E2 -4671.906} C_VEL
LIN {X 0,Y 523.769,Z 409.321,A -85,B 0,C 180,E1 -4672.873,E2 -4672.873} C_VEL
LIN {X 0,Y 523.712,Z 416.154,A -85,B 0,C 180,E1 -4673.84,E2 -4673.84} C_VEL
LIN {X 0,Y 523.488,Z 420.636,A -85,B 0,C 180,E1 -4674.61,E2 -4674.61} C_VEL
LIN {X 0,Y 523.552,Z 424.348,A -85,B 0,C 180,E1 -4675.383,E2 -4675.383} C_VEL
LIN {X 0,Y 523.484,Z 428.586,A -85,B 0,C 180,E1 -4676.539,E2 -4676.539} C_VEL
LIN {X 0,Y 523.338,Z 431.547,A -85,B 0,C 180,E1 -4677.694,E2 -4677.694} C_VEL
LIN {X 0,Y 523.277,Z 432.861,A -85,B 0,C 180,E1 -4678.463,E2 -4678.463} C_VEL
LIN {X 0,Y 523.263,Z 433.679,A -85,B 0,C 180,E1 -4679.233,E2 -4679.233} C_VEL
LIN {X 0,Y 523.265,Z 433.949,A -85,B 0,C 180,E1 -4680.002,E2 -4680.002} C_VEL
LIN {X 0,Y 523.264,Z 433.738,A -85,B 0,C 180,E1 -4680.772,E2 -4680.772} C_VEL
LIN {X 0,Y 523.277,Z 432.99,A -85,B 0,C 180,E1 -4681.542,E2 -4681.542} C_VEL
LIN {X 0,Y 523.34,Z 431.755,A -85,B 0,C 180,E1 -4682.311,E2 -4682.311} C_VEL
LIN {X 0,Y 523.483,Z 428.888,A -85,B 0,C 180,E1 -4683.466,E2 -4683.466} C_VEL
LIN {X 0,Y 523.546,Z 424.77,A -85,B 0,C 180,E1 -4684.622,E2 -4684.622} C_VEL
LIN {X 0,Y 523.61,Z 419.038,A -85,B 0,C 180,E1 -4685.78,E2 -4685.78} C_VEL
LIN {X 0,Y 523.67,Z 413.087,A -85,B 0,C 180,E1 -4686.718,E2 -4686.718} C_VEL
LIN {X 0,Y 523.792,Z 406.844,A -85,B 0,C 180,E1 -4687.519,E2 -4687.519} C_VEL
LIN {X 0,Y 523.987,Z 398.516,A -85,B 0,C 180,E1 -4688.389,E2 -4688.389} C_VEL
LIN {X 0,Y 524.167,Z 388.976,A -85,B 0,C 180,E1 -4689.164,E2 -4689.164} C_VEL
LIN {X 0,Y 524.329,Z 379.823,A -85,B 0,C 180,E1 -4689.745,E2 -4689.745} C_VEL
LIN {X 0,Y 524.432,Z 369.966,A -85,B 0,C 180,E1 -4690.23,E2 -4690.23} C_VEL
LIN {X 0,Y 524.596,Z 358.151,A -85,B 0,C 180,E1 -4690.642,E2 -4690.642} C_VEL
LIN {X 0,Y 524.752,Z 346.201,A -85,B 0,C 180,E1 -4690.882,E2 -4690.882} C_VEL
LIN {X 0,Y 524.761,Z 282.42,A -85,B 0,C 180,E1 -4691.796,E2 -4691.796} C_VEL
LIN {X 0,Y 523.776,Z 276.176,A -85,B 0,C 180,E1 -4691.913,E2 -4691.913} C_VEL
LIN {X 0,Y 523.833,Z 265.684,A -85,B 0,C 180,E1 -4694.373,E2 -4694.373} C_VEL
LIN {X 0,Y 523.947,Z 255.034,A -85,B 0,C 180,E1 -4696.814,E2 -4696.814} C_VEL
LIN {X 0,Y 523.987,Z 255.032,A -85,B 0,C 180,E1 -4700.135,E2 -4700.135} C_VEL
LIN {X 0,Y 523.917,Z 255.034,A -85,B 0,C 180,E1 -4702.895,E2 -4702.895} C_VEL
LIN {X 0,Y 523.908,Z 255.034,A -85,B 0,C 180,E1 -4705.423,E2 -4705.423} C_VEL
LIN {X 0,Y 523.923,Z 255.036,A -85,B 0,C 180,E1 -4708.003,E2 -4708.003} C_VEL
LIN {X 0,Y 523.943,Z 255.032,A -85,B 0,C 180,E1 -4710.854,E2 -4710.854} C_VEL
LIN {X 0,Y 523.937,Z 255.03,A -85,B 0,C 180,E1 -4713.73,E2 -4713.73} C_VEL
LIN {X 0,Y 523.906,Z 255.041,A -85,B 0,C 180,E1 -4716.401,E2 -4716.401} C_VEL
LIN {X 0,Y 523.92,Z 255.033,A -85,B 0,C 180,E1 -4719.086,E2 -4719.086} C_VEL
LIN {X 0,Y 523.948,Z 255.031,A -85,B 0,C 180,E1 -4722.121,E2 -4722.121} C_VEL
LIN {X 0,Y 523.949,Z 255.027,A -85,B 0,C 180,E1 -4725.311,E2 -4725.311} C_VEL
LIN {X 0,Y 523.947,Z 255.035,A -85,B 0,C 180,E1 -4728.692,E2 -4728.692} C_VEL
LIN {X 0,Y 523.919,Z 255.032,A -85,B 0,C 180,E1 -4731.898,E2 -4731.898} C_VEL
LIN {X 0,Y 523.928,Z 255.035,A -85,B 0,C 180,E1 -4734.912,E2 -4734.912} C_VEL
LIN {X 0,Y 523.941,Z 255.029,A -85,B 0,C 180,E1 -4737.68,E2 -4737.68} C_VEL
LIN {X 0,Y 523.959,Z 255.033,A -85,B 0,C 180,E1 -4740.677,E2 -4740.677} C_VEL
LIN {X 0,Y 523.978,Z 255.025,A -85,B 0,C 180,E1 -4743.729,E2 -4743.729} C_VEL
LIN {X 0,Y 523.987,Z 255.205,A -85,B 0,C 180,E1 -4746.692,E2 -4746.692} C_VEL
LIN {X 0,Y 524.855,Z 261.054,A -85,B 0,C 180,E1 -4747.759,E2 -4747.759} C_VEL
LIN {X 0,Y 524.56,Z 275.256,A -85,B 0,C 180,E1 -4750.234,E2 -4750.234} C_VEL
LIN {X 0,Y 524.302,Z 290.437,A -85,B 0,C 180,E1 -4752.848,E2 -4752.848} C_VEL
LIN {X 0,Y 524.004,Z 309.135,A -85,B 0,C 180,E1 -4756.03,E2 -4756.03} C_VEL
LIN {X 0,Y 523.835,Z 321.267,A -85,B 0,C 180,E1 -4758.077,E2 -4758.077} C_VEL
LIN {X 0,Y 524.946,Z 331.849,A -85,B 0,C 180,E1 -4758.253,E2 -4758.253} C_VEL
LIN {X 0,Y 524.69,Z 399.113,A -85,B 0,C 180,E1 -4759.192,E2 -4759.192} C_VEL
LIN {X 0,Y 524.522,Z 408.816,A -85,B 0,C 180,E1 -4759.432,E2 -4759.432} C_VEL
LIN {X 0,Y 524.376,Z 420.419,A -85,B 0,C 180,E1 -4759.868,E2 -4759.868} C_VEL
LIN {X 0,Y 524.189,Z 431.087,A -85,B 0,C 180,E1 -4760.449,E2 -4760.449} C_VEL
LIN {X 0,Y 524.062,Z 439.44,A -85,B 0,C 180,E1 -4761.031,E2 -4761.031} C_VEL
LIN {X 0,Y 523.868,Z 447.342,A -85,B 0,C 180,E1 -4761.708,E2 -4761.708} C_VEL
LIN {X 0,Y 523.702,Z 454.733,A -85,B 0,C 180,E1 -4762.481,E2 -4762.481} C_VEL
LIN {X 0,Y 523.593,Z 461.549,A -85,B 0,C 180,E1 -4763.355,E2 -4763.355} C_VEL
LIN {X 0,Y 523.511,Z 468.124,A -85,B 0,C 180,E1 -4764.414,E2 -4764.414} C_VEL
LIN {X 0,Y 523.402,Z 472.759,A -85,B 0,C 180,E1 -4765.379,E2 -4765.379} C_VEL
LIN {X 0,Y 523.451,Z 475.774,A -85,B 0,C 180,E1 -4766.151,E2 -4766.151} C_VEL
LIN {X 0,Y 523.38,Z 478.108,A -85,B 0,C 180,E1 -4766.921,E2 -4766.921} C_VEL
LIN {X 0,Y 523.337,Z 479.864,A -85,B 0,C 180,E1 -4767.691,E2 -4767.691} C_VEL
LIN {X 0,Y 523.274,Z 481.121,A -85,B 0,C 180,E1 -4768.461,E2 -4768.461} C_VEL
LIN {X 0,Y 523.254,Z 481.904,A -85,B 0,C 180,E1 -4769.23,E2 -4769.23} C_VEL
LIN {X 0,Y 523.257,Z 482.199,A -85,B 0,C 180,E1 -4770,E2 -4770} C_VEL
LIN {X 0,Y 523.254,Z 481.901,A -85,B 0,C 180,E1 -4770.769,E2 -4770.769} C_VEL
LIN {X 0,Y 523.274,Z 481.116,A -85,B 0,C 180,E1 -4771.539,E2 -4771.539} C_VEL
LIN {X 0,Y 523.337,Z 479.857,A -85,B 0,C 180,E1 -4772.309,E2 -4772.309} C_VEL
LIN {X 0,Y 523.406,Z 476.939,A -85,B 0,C 180,E1 -4773.464,E2 -4773.464} C_VEL
LIN {X 0,Y 523.449,Z 474.278,A -85,B 0,C 180,E1 -4774.235,E2 -4774.235} C_VEL
LIN {X 0,Y 523.483,Z 469.069,A -85,B 0,C 180,E1 -4775.392,E2 -4775.392} C_VEL
LIN {X 0,Y 523.578,Z 463.157,A -85,B 0,C 180,E1 -4776.409,E2 -4776.409} C_VEL
LIN {X 0,Y 523.701,Z 456.419,A -85,B 0,C 180,E1 -4777.324,E2 -4777.324} C_VEL
LIN {X 0,Y 523.852,Z 448.349,A -85,B 0,C 180,E1 -4778.195,E2 -4778.195} C_VEL
LIN {X 0,Y 524.055,Z 440.649,A -85,B 0,C 180,E1 -4778.872,E2 -4778.872} C_VEL
LIN {X 0,Y 524.151,Z 432.56,A -85,B 0,C 180,E1 -4779.454,E2 -4779.454} C_VEL
LIN {X 0,Y 524.325,Z 424.185,A -85,B 0,C 180,E1 -4779.937,E2 -4779.937} C_VEL
LIN {X 0,Y 524.446,Z 415.638,A -85,B 0,C 180,E1 -4780.325,E2 -4780.325} C_VEL
LIN {X 0,Y 524.582,Z 406.285,A -85,B 0,C 180,E1 -4780.64,E2 -4780.64} C_VEL
LIN {X 0,Y 524.77,Z 395.188,A -85,B 0,C 180,E1 -4780.88,E2 -4780.88} C_VEL
LIN {X 0,Y 524.79,Z 329.196,A -85,B 0,C 180,E1 -4781.786,E2 -4781.786} C_VEL
LIN {X 0,Y 523.811,Z 321.143,A -85,B 0,C 180,E1 -4781.93,E2 -4781.93} C_VEL
LIN {X 0,Y 524.029,Z 304.304,A -85,B 0,C 180,E1 -4784.763,E2 -4784.763} C_VEL
LIN {X 0,Y 524.398,Z 284.296,A -85,B 0,C 180,E1 -4788.155,E2 -4788.155} C_VEL
LIN {X 0,Y 524.71,Z 266.559,A -85,B 0,C 180,E1 -4791.201,E2 -4791.201} C_VEL
LIN {X 0,Y 524.686,Z 259.418,A -85,B 0,C 180,E1 -4792.446,E2 -4792.446} C_VEL
LIN {X 0,Y 523.958,Z 255.035,A -85,B 0,C 180,E1 -4793.257,E2 -4793.257} C_VEL
LIN {X 0,Y 523.977,Z 255.025,A -85,B 0,C 180,E1 -4796.271,E2 -4796.271} C_VEL
LIN {X 0,Y 523.958,Z 255.033,A -85,B 0,C 180,E1 -4799.323,E2 -4799.323} C_VEL
LIN {X 0,Y 523.938,Z 255.027,A -85,B 0,C 180,E1 -4802.449,E2 -4802.449} C_VEL
LIN {X 0,Y 523.924,Z 255.038,A -85,B 0,C 180,E1 -4805.226,E2 -4805.226} C_VEL
LIN {X 0,Y 523.918,Z 255.032,A -85,B 0,C 180,E1 -4808.101,E2 -4808.101} C_VEL
LIN {X 0,Y 523.944,Z 255.032,A -85,B 0,C 180,E1 -4811.092,E2 -4811.092} C_VEL
LIN {X 0,Y 523.935,Z 255.028,A -85,B 0,C 180,E1 -4814.228,E2 -4814.228} C_VEL
LIN {X 0,Y 523.922,Z 255.031,A -85,B 0,C 180,E1 -4816.832,E2 -4816.832} C_VEL
LIN {X 0,Y 523.944,Z 255.029,A -85,B 0,C 180,E1 -4818.907,E2 -4818.907} C_VEL
LIN {X 0,Y 523.92,Z 255.035,A -85,B 0,C 180,E1 -4821.897,E2 -4821.897} C_VEL
LIN {X 0,Y 523.929,Z 255.028,A -85,B 0,C 180,E1 -4824.91,E2 -4824.91} C_VEL
LIN {X 0,Y 523.941,Z 255.036,A -85,B 0,C 180,E1 -4827.679,E2 -4827.679} C_VEL
LIN {X 0,Y 523.957,Z 255.025,A -85,B 0,C 180,E1 -4830.676,E2 -4830.676} C_VEL
LIN {X 0,Y 523.943,Z 255.034,A -85,B 0,C 180,E1 -4833.725,E2 -4833.725} C_VEL
LIN {X 0,Y 523.917,Z 255.033,A -85,B 0,C 180,E1 -4836.268,E2 -4836.268} C_VEL
LIN {X 0,Y 523.951,Z 255.023,A -85,B 0,C 180,E1 -4838.765,E2 -4838.765} C_VEL
LIN {X 0,Y 523.943,Z 255.029,A -85,B 0,C 180,E1 -4841.219,E2 -4841.219} C_VEL
LIN {X 0,Y 523.932,Z 255.033,A -85,B 0,C 180,E1 -4843.637,E2 -4843.637} C_VEL
LIN {X 0,Y 523.94,Z 255.035,A -85,B 0,C 180,E1 -4846.026,E2 -4846.026} C_VEL
LIN {X 0,Y 523.997,Z 255.017,A -85,B 0,C 180,E1 -4849.175,E2 -4849.175} C_VEL
LIN {X 0,Y 524.031,Z 255.019,A -85,B 0,C 180,E1 -4852.29,E2 -4852.29} C_VEL
LIN {X 0,Y 524.08,Z 255.008,A -85,B 0,C 180,E1 -4854.611,E2 -4854.611} C_VEL
LIN {X 0,Y 524.112,Z 255.009,A -85,B 0,C 180,E1 -4857.692,E2 -4857.692} C_VEL
LIN {X 0,Y 524.118,Z 255.005,A -85,B 0,C 180,E1 -4860.766,E2 -4860.766} C_VEL
LIN {X 0,Y 524.039,Z 255.014,A -85,B 0,C 180,E1 -4863.073,E2 -4863.073} C_VEL
LIN {X 0,Y 524.022,Z 255.023,A -85,B 0,C 180,E1 -4866.157,E2 -4866.157} C_VEL
LIN {X 0,Y 523.984,Z 255.021,A -85,B 0,C 180,E1 -4869.259,E2 -4869.259} C_VEL
LIN {X 0,Y 523.998,Z 255.021,A -85,B 0,C 180,E1 -4871.736,E2 -4871.736} C_VEL
LIN {X 0,Y 523.987,Z 255.021,A -85,B 0,C 180,E1 -4875.049,E2 -4875.049} C_VEL
LIN {X 0,Y 523.939,Z 255.032,A -85,B 0,C 180,E1 -4877.967,E2 -4877.967} C_VEL
LIN {X 0,Y 523.962,Z 255.032,A -85,B 0,C 180,E1 -4880.407,E2 -4880.407} C_VEL
LIN {X 0,Y 523.899,Z 255.035,A -85,B 0,C 180,E1 -4882.891,E2 -4882.891} C_VEL
LIN {X 0,Y 523.94,Z 255.027,A -85,B 0,C 180,E1 -4885.416,E2 -4885.416} C_VEL
LIN {X 0,Y 523.956,Z 255.028,A -85,B 0,C 180,E1 -4887.996,E2 -4887.996} C_VEL
LIN {X 0,Y 523.929,Z 255.033,A -85,B 0,C 180,E1 -4890.852,E2 -4890.852} C_VEL
LIN {X 0,Y 523.943,Z 255.028,A -85,B 0,C 180,E1 -4893.732,E2 -4893.732} C_VEL
LIN {X 0,Y 523.9,Z 255.036,A -85,B 0,C 180,E1 -4896.401,E2 -4896.401} C_VEL
LIN {X 0,Y 523.9,Z 255.035,A -85,B 0,C 180,E1 -4899.082,E2 -4899.082} C_VEL
LIN {X 0,Y 523.935,Z 255.031,A -85,B 0,C 180,E1 -4902.115,E2 -4902.115} C_VEL
LIN {X 0,Y 523.93,Z 255.032,A -85,B 0,C 180,E1 -4905.306,E2 -4905.306} C_VEL
LIN {X 0,Y 523.898,Z 255.04,A -85,B 0,C 180,E1 -4906.89,E2 -4906.89} C_VEL
LIN {X 0,Y 523.233,Z 255.119,A -85,B 0,C 180,E1 -4907.531,E2 -4907.531} C_VEL
LIN {X 0,Y 520.398,Z 255.477,A -85,B 0,C 180,E1 -4908.573,E2 -4908.573} C_VEL
LIN {X 0,Y 518.001,Z 255.773,A -85,B 0,C 180,E1 -4909.412,E2 -4909.412} C_VEL
LIN {X 0,Y 516.969,Z 255.9,A -85,B 0,C 180,E1 -4910.06,E2 -4910.06} C_VEL
LIN {X 0,Y 516.884,Z 255.911,A -85,B 0,C 180,E1 -4910.279,E2 -4910.279} C_VEL
LIN {X 0,Y 516.857,Z 255.915,A -85,B 0,C 180,E1 -4913.339,E2 -4913.339} C_VEL
LIN {X 0,Y 516.892,Z 255.912,A -85,B 0,C 180,E1 -4916.354,E2 -4916.354} C_VEL
LIN {X 0,Y 516.771,Z 255.963,A -85,B 0,C 180,E1 -4916.579,E2 -4916.579} C_VEL
LIN {X 0,Y 516.705,Z 266.885,A -85,B 0,C 180,E1 -4918.962,E2 -4918.962} C_VEL
LIN {X 0,Y 516.727,Z 276.026,A -85,B 0,C 180,E1 -4920.978,E2 -4920.978} C_VEL
LIN {X 0,Y 518.086,Z 284.879,A -85,B 0,C 180,E1 -4921.141,E2 -4921.141} C_VEL
LIN {X 0,Y 517.772,Z 352.023,A -85,B 0,C 180,E1 -4922.092,E2 -4922.092} C_VEL
LIN {X 0,Y 517.668,Z 362.168,A -85,B 0,C 180,E1 -4922.352,E2 -4922.352} C_VEL
LIN {X 0,Y 517.506,Z 374.214,A -85,B 0,C 180,E1 -4922.829,E2 -4922.829} C_VEL
LIN {X 0,Y 517.342,Z 383.775,A -85,B 0,C 180,E1 -4923.366,E2 -4923.366} C_VEL
LIN {X 0,Y 517.194,Z 391.71,A -85,B 0,C 180,E1 -4923.926,E2 -4923.926} C_VEL
LIN {X 0,Y 516.966,Z 398.851,A -85,B 0,C 180,E1 -4924.537,E2 -4924.537} C_VEL
LIN {X 0,Y 516.809,Z 405.63,A -85,B 0,C 180,E1 -4925.238,E2 -4925.238} C_VEL
LIN {X 0,Y 516.725,Z 411.158,A -85,B 0,C 180,E1 -4925.919,E2 -4925.919} C_VEL
LIN {X 0,Y 516.576,Z 416.861,A -85,B 0,C 180,E1 -4926.763,E2 -4926.763} C_VEL
LIN {X 0,Y 516.466,Z 422.041,A -85,B 0,C 180,E1 -4927.707,E2 -4927.707} C_VEL
LIN {X 0,Y 516.371,Z 426.96,A -85,B 0,C 180,E1 -4928.858,E2 -4928.858} C_VEL
LIN {X 0,Y 516.332,Z 430.797,A -85,B 0,C 180,E1 -4930.106,E2 -4930.106} C_VEL
LIN {X 0,Y 516.223,Z 432.504,A -85,B 0,C 180,E1 -4930.929,E2 -4930.929} C_VEL
LIN {X 0,Y 516.224,Z 434.085,A -85,B 0,C 180,E1 -4932.348,E2 -4932.348} C_VEL
LIN {X 0,Y 516.215,Z 434.227,A -85,B 0,C 180,E1 -4933.387,E2 -4933.387} C_VEL
LIN {X 0,Y 516.246,Z 433.768,A -85,B 0,C 180,E1 -4934.201,E2 -4934.201} C_VEL
LIN {X 0,Y 516.248,Z 432.565,A -85,B 0,C 180,E1 -4935.125,E2 -4935.125} C_VEL
LIN {X 0,Y 516.335,Z 430.137,A -85,B 0,C 180,E1 -4936.22,E2 -4936.22} C_VEL
LIN {X 0,Y 516.371,Z 427.734,A -85,B 0,C 180,E1 -4937.022,E2 -4937.022} C_VEL
LIN {X 0,Y 516.446,Z 422.8,A -85,B 0,C 180,E1 -4938.222,E2 -4938.222} C_VEL
LIN {X 0,Y 516.529,Z 418.673,A -85,B 0,C 180,E1 -4939.019,E2 -4939.019} C_VEL
LIN {X 0,Y 516.618,Z 413.704,A -85,B 0,C 180,E1 -4939.814,E2 -4939.814} C_VEL
LIN {X 0,Y 516.78,Z 407.693,A -85,B 0,C 180,E1 -4940.608,E2 -4940.608} C_VEL
LIN {X 0,Y 516.972,Z 400.38,A -85,B 0,C 180,E1 -4941.4,E2 -4941.4} C_VEL
LIN {X 0,Y 517.104,Z 393.819,A -85,B 0,C 180,E1 -4941.992,E2 -4941.992} C_VEL
LIN {X 0,Y 517.301,Z 385.489,A -85,B 0,C 180,E1 -4942.609,E2 -4942.609} C_VEL
LIN {X 0,Y 517.435,Z 377.66,A -85,B 0,C 180,E1 -4943.077,E2 -4943.077} C_VEL
LIN {X 0,Y 517.549,Z 369.365,A -85,B 0,C 180,E1 -4943.47,E2 -4943.47} C_VEL
LIN {X 0,Y 517.664,Z 360.39,A -85,B 0,C 180,E1 -4943.789,E2 -4943.789} C_VEL
LIN {X 0,Y 517.768,Z 351.288,A -85,B 0,C 180,E1 -4944.011,E2 -4944.011} C_VEL
LIN {X 0,Y 517.882,Z 283.192,A -85,B 0,C 180,E1 -4944.976,E2 -4944.976} C_VEL
LIN {X 0,Y 516.765,Z 276.049,A -85,B 0,C 180,E1 -4945.124,E2 -4945.124} C_VEL
LIN {X 0,Y 516.865,Z 261.563,A -85,B 0,C 180,E1 -4948.442,E2 -4948.442} C_VEL
LIN {X 0,Y 516.868,Z 255.914,A -85,B 0,C 180,E1 -4949.757,E2 -4949.757} C_VEL
LIN {X 0,Y 517.058,Z 255.891,A -85,B 0,C 180,E1 -4950.779,E2 -4950.779} C_VEL
LIN {X 0,Y 516.98,Z 255.902,A -85,B 0,C 180,E1 -4953.117,E2 -4953.117} C_VEL
LIN {X 0,Y 516.965,Z 255.897,A -85,B 0,C 180,E1 -4956.244,E2 -4956.244} C_VEL
LIN {X 0,Y 516.915,Z 255.911,A -85,B 0,C 180,E1 -4959.39,E2 -4959.39} C_VEL
LIN {X 0,Y 516.919,Z 255.905,A -85,B 0,C 180,E1 -4961.811,E2 -4961.811} C_VEL
LIN {X 0,Y 516.905,Z 255.91,A -85,B 0,C 180,E1 -4965.147,E2 -4965.147} C_VEL
LIN {X 0,Y 516.887,Z 255.907,A -85,B 0,C 180,E1 -4968.224,E2 -4968.224} C_VEL
LIN {X 0,Y 516.875,Z 255.909,A -85,B 0,C 180,E1 -4970.703,E2 -4970.703} C_VEL
LIN {X 0,Y 516.85,Z 255.912,A -85,B 0,C 180,E1 -4974.075,E2 -4974.075} C_VEL
LIN {X 0,Y 516.86,Z 255.91,A -85,B 0,C 180,E1 -4976.662,E2 -4976.662} C_VEL
LIN {X 0,Y 516.875,Z 255.917,A -85,B 0,C 180,E1 -4979.525,E2 -4979.525} C_VEL
LIN {X 0,Y 516.864,Z 255.909,A -85,B 0,C 180,E1 -4982.546,E2 -4982.546} C_VEL
LIN {X 0,Y 516.833,Z 255.919,A -85,B 0,C 180,E1 -4985.332,E2 -4985.332} C_VEL
LIN {X 0,Y 516.848,Z 255.915,A -85,B 0,C 180,E1 -4987.945,E2 -4987.945} C_VEL
LIN {X 0,Y 516.837,Z 255.913,A -85,B 0,C 180,E1 -4990.746,E2 -4990.746} C_VEL
LIN {X 0,Y 516.833,Z 255.914,A -85,B 0,C 180,E1 -4992.837,E2 -4992.837} C_VEL
LIN {X 0,Y 516.871,Z 255.91,A -85,B 0,C 180,E1 -4995.01,E2 -4995.01} C_VEL
LIN {X 0,Y 516.892,Z 255.907,A -85,B 0,C 180,E1 -4998.402,E2 -4998.402} C_VEL
LIN {X 0,Y 516.859,Z 255.914,A -85,B 0,C 180,E1 -5001.287,E2 -5001.287} C_VEL
LIN {X 0,Y 516.852,Z 255.913,A -85,B 0,C 180,E1 -5004.223,E2 -5004.223} C_VEL
LIN {X 0,Y 516.865,Z 255.911,A -85,B 0,C 180,E1 -5007.055,E2 -5007.055} C_VEL
LIN {X 0,Y 516.877,Z 255.917,A -85,B 0,C 180,E1 -5009.799,E2 -5009.799} C_VEL
LIN {X 0,Y 516.879,Z 255.909,A -85,B 0,C 180,E1 -5012.468,E2 -5012.468} C_VEL
LIN {X 0,Y 516.85,Z 255.912,A -85,B 0,C 180,E1 -5015.073,E2 -5015.073} C_VEL
LIN {X 0,Y 516.86,Z 255.916,A -85,B 0,C 180,E1 -5017.625,E2 -5017.625} C_VEL
LIN {X 0,Y 516.921,Z 255.907,A -85,B 0,C 180,E1 -5020.133,E2 -5020.133} C_VEL
LIN {X 0,Y 516.908,Z 255.964,A -85,B 0,C 180,E1 -5023.261,E2 -5023.261} C_VEL
LIN {X 0,Y 516.811,Z 266.878,A -85,B 0,C 180,E1 -5025.834,E2 -5025.834} C_VEL
LIN {X 0,Y 516.705,Z 276.152,A -85,B 0,C 180,E1 -5028.011,E2 -5028.011} C_VEL
LIN {X 0,Y 518.007,Z 285.276,A -85,B 0,C 180,E1 -5028.179,E2 -5028.179} C_VEL
LIN {X 0,Y 517.684,Z 352.413,A -85,B 0,C 180,E1 -5029.17,E2 -5029.17} C_VEL
LIN {X 0,Y 517.568,Z 362.436,A -85,B 0,C 180,E1 -5029.44,E2 -5029.44} C_VEL
LIN {X 0,Y 517.42,Z 371.346,A -85,B 0,C 180,E1 -5029.783,E2 -5029.783} C_VEL
LIN {X 0,Y 517.298,Z 380.06,A -85,B 0,C 180,E1 -5030.225,E2 -5030.225} C_VEL
LIN {X 0,Y 517.174,Z 389.184,A -85,B 0,C 180,E1 -5030.815,E2 -5030.815} C_VEL
LIN {X 0,Y 516.953,Z 398.703,A -85,B 0,C 180,E1 -5031.599,E2 -5031.599} C_VEL
LIN {X 0,Y 516.773,Z 406.207,A -85,B 0,C 180,E1 -5032.383,E2 -5032.383} C_VEL
LIN {X 0,Y 516.66,Z 412.764,A -85,B 0,C 180,E1 -5033.219,E2 -5033.219} C_VEL
LIN {X 0,Y 516.568,Z 418.689,A -85,B 0,C 180,E1 -5034.146,E2 -5034.146} C_VEL
LIN {X 0,Y 516.426,Z 422.767,A -85,B 0,C 180,E1 -5034.928,E2 -5034.928} C_VEL
LIN {X 0,Y 516.433,Z 426.123,A -85,B 0,C 180,E1 -5035.71,E2 -5035.71} C_VEL
LIN {X 0,Y 516.403,Z 429.995,A -85,B 0,C 180,E1 -5036.882,E2 -5036.882} C_VEL
LIN {X 0,Y 516.267,Z 431.832,A -85,B 0,C 180,E1 -5037.662,E2 -5037.662} C_VEL
LIN {X 0,Y 516.194,Z 433.153,A -85,B 0,C 180,E1 -5038.442,E2 -5038.442} C_VEL
LIN {X 0,Y 516.172,Z 433.984,A -85,B 0,C 180,E1 -5039.222,E2 -5039.222} C_VEL
LIN {X 0,Y 516.174,Z 434.283,A -85,B 0,C 180,E1 -5040.003,E2 -5040.003} C_VEL
LIN {X 0,Y 516.173,Z 434.038,A -85,B 0,C 180,E1 -5040.783,E2 -5040.783} C_VEL
LIN {X 0,Y 516.194,Z 433.288,A -85,B 0,C 180,E1 -5041.563,E2 -5041.563} C_VEL
LIN {X 0,Y 516.269,Z 432.05,A -85,B 0,C 180,E1 -5042.343,E2 -5042.343} C_VEL
LIN {X 0,Y 516.419,Z 429.179,A -85,B 0,C 180,E1 -5043.513,E2 -5043.513} C_VEL
LIN {X 0,Y 516.469,Z 425.052,A -85,B 0,C 180,E1 -5044.686,E2 -5044.686} C_VEL
LIN {X 0,Y 516.563,Z 419.276,A -85,B 0,C 180,E1 -5045.859,E2 -5045.859} C_VEL
LIN {X 0,Y 516.621,Z 413.754,A -85,B 0,C 180,E1 -5046.744,E2 -5046.744} C_VEL
LIN {X 0,Y 516.752,Z 408.661,A -85,B 0,C 180,E1 -5047.426,E2 -5047.426} C_VEL
LIN {X 0,Y 516.857,Z 401.607,A -85,B 0,C 180,E1 -5048.211,E2 -5048.211} C_VEL
LIN {X 0,Y 517.044,Z 394.086,A -85,B 0,C 180,E1 -5048.897,E2 -5048.897} C_VEL
LIN {X 0,Y 517.276,Z 384.79,A -85,B 0,C 180,E1 -5049.583,E2 -5049.583} C_VEL
LIN {X 0,Y 517.422,Z 374.257,A -85,B 0,C 180,E1 -5050.173,E2 -5050.173} C_VEL
LIN {X 0,Y 517.547,Z 364.002,A -85,B 0,C 180,E1 -5050.59,E2 -5050.59} C_VEL
LIN {X 0,Y 517.623,Z 354.519,A -85,B 0,C 180,E1 -5050.861,E2 -5050.861} C_VEL
LIN {X 0,Y 517.77,Z 340.613,A -85,B 0,C 180,E1 -5051.097,E2 -5051.097} C_VEL
LIN {X 0,Y 517.817,Z 283.084,A -85,B 0,C 180,E1 -5051.944,E2 -5051.944} C_VEL
LIN {X 0,Y 516.715,Z 276.562,A -85,B 0,C 180,E1 -5052.072,E2 -5052.072} C_VEL
LIN {X 0,Y 516.85,Z 263.385,A -85,B 0,C 180,E1 -5055.106,E2 -5055.106} C_VEL
LIN {X 0,Y 516.908,Z 255.912,A -85,B 0,C 180,E1 -5056.846,E2 -5056.846} C_VEL
LIN {X 0,Y 516.937,Z 255.909,A -85,B 0,C 180,E1 -5059.872,E2 -5059.872} C_VEL
LIN {X 0,Y 516.874,Z 255.918,A -85,B 0,C 180,E1 -5062.391,E2 -5062.391} C_VEL
LIN {X 0,Y 516.854,Z 255.914,A -85,B 0,C 180,E1 -5064.933,E2 -5064.933} C_VEL
LIN {X 0,Y 516.886,Z 255.911,A -85,B 0,C 180,E1 -5067.896,E2 -5067.896} C_VEL
LIN {X 0,Y 516.891,Z 255.914,A -85,B 0,C 180,E1 -5070.205,E2 -5070.205} C_VEL
LIN {X 0,Y 516.889,Z 255.91,A -85,B 0,C 180,E1 -5072.949,E2 -5072.949} C_VEL
LIN {X 0,Y 516.875,Z 255.91,A -85,B 0,C 180,E1 -5075.782,E2 -5075.782} C_VEL
LIN {X 0,Y 516.884,Z 255.914,A -85,B 0,C 180,E1 -5078.717,E2 -5078.717} C_VEL
LIN {X 0,Y 516.91,Z 255.905,A -85,B 0,C 180,E1 -5081.777,E2 -5081.777} C_VEL
LIN {X 0,Y 516.903,Z 255.908,A -85,B 0,C 180,E1 -5085.007,E2 -5085.007} C_VEL
LIN {X 0,Y 516.91,Z 255.91,A -85,B 0,C 180,E1 -5088.401,E2 -5088.401} C_VEL
LIN {X 0,Y 516.885,Z 255.908,A -85,B 0,C 180,E1 -5091.284,E2 -5091.284} C_VEL
LIN {X 0,Y 516.874,Z 255.91,A -85,B 0,C 180,E1 -5094.22,E2 -5094.22} C_VEL
LIN {X 0,Y 516.887,Z 255.911,A -85,B 0,C 180,E1 -5097.052,E2 -5097.052} C_VEL
LIN {X 0,Y 516.892,Z 255.907,A -85,B 0,C 180,E1 -5099.796,E2 -5099.796} C_VEL
LIN {X 0,Y 516.929,Z 255.908,A -85,B 0,C 180,E1 -5102.467,E2 -5102.467} C_VEL
LIN {X 0,Y 516.877,Z 255.916,A -85,B 0,C 180,E1 -5105.07,E2 -5105.07} C_VEL
LIN {X 0,Y 516.958,Z 256.057,A -85,B 0,C 180,E1 -5106.568,E2 -5106.568} C_VEL
LIN {X 0,Y 517.85,Z 261.987,A -85,B 0,C 180,E1 -5107.666,E2 -5107.666} C_VEL
LIN {X 0,Y 517.641,Z 274.248,A -85,B 0,C 180,E1 -5109.835,E2 -5109.835} C_VEL
LIN {X 0,Y 517.311,Z 290.132,A -85,B 0,C 180,E1 -5112.609,E2 -5112.609} C_VEL
LIN {X 0,Y 516.977,Z 308.814,A -85,B 0,C 180,E1 -5115.836,E2 -5115.836} C_VEL
LIN {X 0,Y 516.779,Z 320.942,A -85,B 0,C 180,E1 -5117.911,E2 -5117.911} C_VEL
LIN {X 0,Y 517.986,Z 331.529,A -85,B 0,C 180,E1 -5118.093,E2 -5118.093} C_VEL
LIN {X 0,Y 517.723,Z 398.75,A -85,B 0,C 180,E1 -5119.044,E2 -5119.044} C_VEL
LIN {X 0,Y 517.551,Z 408.468,A -85,B 0,C 180,E1 -5119.288,E2 -5119.288} C_VEL
LIN {X 0,Y 517.38,Z 420.079,A -85,B 0,C 180,E1 -5119.73,E2 -5119.73} C_VEL
LIN {X 0,Y 517.17,Z 430.751,A -85,B 0,C 180,E1 -5120.318,E2 -5120.318} C_VEL
LIN {X 0,Y 517.009,Z 439.106,A -85,B 0,C 180,E1 -5120.908,E2 -5120.908} C_VEL
LIN {X 0,Y 516.821,Z 447.011,A -85,B 0,C 180,E1 -5121.594,E2 -5121.594} C_VEL
LIN {X 0,Y 516.652,Z 454.403,A -85,B 0,C 180,E1 -5122.378,E2 -5122.378} C_VEL
LIN {X 0,Y 516.515,Z 461.9,A -85,B 0,C 180,E1 -5123.358,E2 -5123.358} C_VEL
LIN {X 0,Y 516.438,Z 467.797,A -85,B 0,C 180,E1 -5124.338,E2 -5124.338} C_VEL
LIN {X 0,Y 516.31,Z 472.432,A -85,B 0,C 180,E1 -5125.315,E2 -5125.315} C_VEL
LIN {X 0,Y 516.362,Z 475.448,A -85,B 0,C 180,E1 -5126.098,E2 -5126.098} C_VEL
LIN {X 0,Y 516.295,Z 477.782,A -85,B 0,C 180,E1 -5126.879,E2 -5126.879} C_VEL
LIN {X 0,Y 516.264,Z 479.539,A -85,B 0,C 180,E1 -5127.659,E2 -5127.659} C_VEL
LIN {X 0,Y 516.191,Z 480.795,A -85,B 0,C 180,E1 -5128.439,E2 -5128.439} C_VEL
LIN {X 0,Y 516.163,Z 481.578,A -85,B 0,C 180,E1 -5129.22,E2 -5129.22} C_VEL
LIN {X 0,Y 516.165,Z 481.873,A -85,B 0,C 180,E1 -5130,E2 -5130} C_VEL
LIN {X 0,Y 516.163,Z 481.574,A -85,B 0,C 180,E1 -5130.78,E2 -5130.78} C_VEL
LIN {X 0,Y 516.191,Z 480.788,A -85,B 0,C 180,E1 -5131.56,E2 -5131.56} C_VEL
LIN {X 0,Y 516.263,Z 479.529,A -85,B 0,C 180,E1 -5132.34,E2 -5132.34} C_VEL
LIN {X 0,Y 516.324,Z 476.608,A -85,B 0,C 180,E1 -5133.512,E2 -5133.512} C_VEL
LIN {X 0,Y 516.34,Z 473.945,A -85,B 0,C 180,E1 -5134.293,E2 -5134.293} C_VEL
LIN {X 0,Y 516.421,Z 468.736,A -85,B 0,C 180,E1 -5135.466,E2 -5135.466} C_VEL
LIN {X 0,Y 516.481,Z 463.495,A -85,B 0,C 180,E1 -5136.386,E2 -5136.386} C_VEL
LIN {X 0,Y 516.625,Z 456.08,A -85,B 0,C 180,E1 -5137.425,E2 -5137.425} C_VEL
LIN {X 0,Y 516.806,Z 448.007,A -85,B 0,C 180,E1 -5138.308,E2 -5138.308} C_VEL
LIN {X 0,Y 516.991,Z 440.304,A -85,B 0,C 180,E1 -5138.994,E2 -5138.994} C_VEL
LIN {X 0,Y 517.127,Z 432.213,A -85,B 0,C 180,E1 -5139.583,E2 -5139.583} C_VEL
LIN {X 0,Y 517.302,Z 423.834,A -85,B 0,C 180,E1 -5140.074,E2 -5140.074} C_VEL
LIN {X 0,Y 517.436,Z 415.282,A -85,B 0,C 180,E1 -5140.467,E2 -5140.467} C_VEL
LIN {X 0,Y 517.614,Z 405.924,A -85,B 0,C 180,E1 -5140.784,E2 -5140.784} C_VEL
LIN {X 0,Y 517.801,Z 394.942,A -85,B 0,C 180,E1 -5141.026,E2 -5141.026} C_VEL
LIN {X 0,Y 517.878,Z 330.193,A -85,B 0,C 180,E1 -5141.927,E2 -5141.927} C_VEL
LIN {X 0,Y 516.749,Z 320.78,A -85,B 0,C 180,E1 -5142.1,E2 -5142.1} C_VEL
LIN {X 0,Y 516.989,Z 303.957,A -85,B 0,C 180,E1 -5144.968,E2 -5144.968} C_VEL
LIN {X 0,Y 517.363,Z 285.117,A -85,B 0,C 180,E1 -5148.206,E2 -5148.206} C_VEL
LIN {X 0,Y 517.734,Z 267.401,A -85,B 0,C 180,E1 -5151.292,E2 -5151.292} C_VEL
LIN {X 0,Y 517.617,Z 260.09,A -85,B 0,C 180,E1 -5152.589,E2 -5152.589} C_VEL
LIN {X 0,Y 516.897,Z 255.914,A -85,B 0,C 180,E1 -5153.381,E2 -5153.381} C_VEL
LIN {X 0,Y 516.928,Z 255.905,A -85,B 0,C 180,E1 -5156.658,E2 -5156.658} C_VEL
LIN {X 0,Y 516.913,Z 255.909,A -85,B 0,C 180,E1 -5159.523,E2 -5159.523} C_VEL
LIN {X 0,Y 516.899,Z 255.904,A -85,B 0,C 180,E1 -5162.542,E2 -5162.542} C_VEL
LIN {X 0,Y 516.87,Z 255.915,A -85,B 0,C 180,E1 -5165.329,E2 -5165.329} C_VEL
LIN {X 0,Y 516.884,Z 255.91,A -85,B 0,C 180,E1 -5167.942,E2 -5167.942} C_VEL
LIN {X 0,Y 516.888,Z 255.908,A -85,B 0,C 180,E1 -5170.741,E2 -5170.741} C_VEL
LIN {X 0,Y 516.868,Z 255.911,A -85,B 0,C 180,E1 -5172.833,E2 -5172.833} C_VEL
LIN {X 0,Y 516.901,Z 255.906,A -85,B 0,C 180,E1 -5175.006,E2 -5175.006} C_VEL
LIN {X 0,Y 516.919,Z 255.903,A -85,B 0,C 180,E1 -5178.398,E2 -5178.398} C_VEL
LIN {X 0,Y 516.883,Z 255.911,A -85,B 0,C 180,E1 -5181.283,E2 -5181.283} C_VEL
LIN {X 0,Y 516.877,Z 255.907,A -85,B 0,C 180,E1 -5184.219,E2 -5184.219} C_VEL
LIN {X 0,Y 516.887,Z 255.908,A -85,B 0,C 180,E1 -5187.051,E2 -5187.051} C_VEL
LIN {X 0,Y 516.889,Z 255.914,A -85,B 0,C 180,E1 -5189.794,E2 -5189.794} C_VEL
LIN {X 0,Y 516.903,Z 255.904,A -85,B 0,C 180,E1 -5192.464,E2 -5192.464} C_VEL
LIN {X 0,Y 516.872,Z 255.908,A -85,B 0,C 180,E1 -5195.068,E2 -5195.068} C_VEL
LIN {X 0,Y 516.875,Z 255.915,A -85,B 0,C 180,E1 -5197.62,E2 -5197.62} C_VEL
LIN {X 0,Y 516.935,Z 255.905,A -85,B 0,C 180,E1 -5200.128,E2 -5200.128} C_VEL
LIN {X 0,Y 516.902,Z 255.903,A -85,B 0,C 180,E1 -5202.593,E2 -5202.593} C_VEL
LIN {X 0,Y 516.948,Z 255.897,A -85,B 0,C 180,E1 -5205.028,E2 -5205.028} C_VEL
LIN {X 0,Y 516.97,Z 255.897,A -85,B 0,C 180,E1 -5208.232,E2 -5208.232} C_VEL
LIN {X 0,Y 516.967,Z 255.897,A -85,B 0,C 180,E1 -5211.397,E2 -5211.397} C_VEL
LIN {X 0,Y 517.01,Z 255.895,A -85,B 0,C 180,E1 -5213.755,E2 -5213.755} C_VEL
LIN {X 0,Y 517.082,Z 255.884,A -85,B 0,C 180,E1 -5217.661,E2 -5217.661} C_VEL
LIN {X 0,Y 517.089,Z 255.88,A -85,B 0,C 180,E1 -5220.776,E2 -5220.776} C_VEL
LIN {X 0,Y 516.983,Z 255.893,A -85,B 0,C 180,E1 -5223.114,E2 -5223.114} C_VEL
LIN {X 0,Y 516.985,Z 255.901,A -85,B 0,C 180,E1 -5226.241,E2 -5226.241} C_VEL
LIN {X 0,Y 516.939,Z 255.899,A -85,B 0,C 180,E1 -5229.387,E2 -5229.387} C_VEL
LIN {X 0,Y 516.947,Z 255.9,A -85,B 0,C 180,E1 -5231.804,E2 -5231.804} C_VEL
LIN {X 0,Y 516.938,Z 255.898,A -85,B 0,C 180,E1 -5235.143,E2 -5235.143} C_VEL
LIN {X 0,Y 516.908,Z 255.911,A -85,B 0,C 180,E1 -5238.219,E2 -5238.219} C_VEL
LIN {X 0,Y 516.902,Z 255.908,A -85,B 0,C 180,E1 -5240.698,E2 -5240.698} C_VEL
LIN {X 0,Y 516.891,Z 255.91,A -85,B 0,C 180,E1 -5244.069,E2 -5244.069} C_VEL
LIN {X 0,Y 516.913,Z 255.909,A -85,B 0,C 180,E1 -5246.655,E2 -5246.655} C_VEL
LIN {X 0,Y 516.897,Z 255.905,A -85,B 0,C 180,E1 -5249.521,E2 -5249.521} C_VEL
LIN {X 0,Y 516.88,Z 255.916,A -85,B 0,C 180,E1 -5252.541,E2 -5252.541} C_VEL
LIN {X 0,Y 516.86,Z 255.907,A -85,B 0,C 180,E1 -5255.329,E2 -5255.329} C_VEL
LIN {X 0,Y 516.86,Z 255.911,A -85,B 0,C 180,E1 -5257.94,E2 -5257.94} C_VEL
LIN {X 0,Y 516.874,Z 255.915,A -85,B 0,C 180,E1 -5260.738,E2 -5260.738} C_VEL
LIN {X 0,Y 516.881,Z 255.914,A -85,B 0,C 180,E1 -5262.826,E2 -5262.826} C_VEL
LIN {X 0,Y 516.898,Z 255.911,A -85,B 0,C 180,E1 -5265.007,E2 -5265.007} C_VEL
LIN {X 0,Y 516.902,Z 255.91,A -85,B 0,C 180,E1 -5268.394,E2 -5268.394} C_VEL
LIN {X 0,Y 516.884,Z 255.911,A -85,B 0,C 180,E1 -5270.279,E2 -5270.279} C_VEL
LIN {X 0,Y 516.212,Z 255.999,A -85,B 0,C 180,E1 -5270.929,E2 -5270.929} C_VEL
LIN {X 0,Y 513.357,Z 256.353,A -85,B 0,C 180,E1 -5271.984,E2 -5271.984} C_VEL
LIN {X 0,Y 510.939,Z 256.657,A -85,B 0,C 180,E1 -5272.834,E2 -5272.834} C_VEL
LIN {X 0,Y 509.894,Z 256.782,A -85,B 0,C 180,E1 -5273.49,E2 -5273.49} C_VEL
LIN {X 0,Y 509.805,Z 256.792,A -85,B 0,C 180,E1 -5273.713,E2 -5273.713} C_VEL
LIN {X 0,Y 509.844,Z 256.788,A -85,B 0,C 180,E1 -5275.792,E2 -5275.792} C_VEL
LIN {X 0,Y 509.732,Z 257.012,A -85,B 0,C 180,E1 -5276.579,E2 -5276.579} C_VEL
LIN {X 0,Y 509.688,Z 269.529,A -85,B 0,C 180,E1 -5279.324,E2 -5279.324} C_VEL
LIN {X 0,Y 509.676,Z 276.247,A -85,B 0,C 180,E1 -5280.808,E2 -5280.808} C_VEL
LIN {X 0,Y 511.155,Z 285.915,A -85,B 0,C 180,E1 -5280.988,E2 -5280.988} C_VEL
LIN {X 0,Y 510.81,Z 352.343,A -85,B 0,C 180,E1 -5281.942,E2 -5281.942} C_VEL
LIN {X 0,Y 510.708,Z 361.884,A -85,B 0,C 180,E1 -5282.187,E2 -5282.187} C_VEL
LIN {X 0,Y 510.581,Z 372.62,A -85,B 0,C 180,E1 -5282.596,E2 -5282.596} C_VEL
LIN {X 0,Y 510.365,Z 383.864,A -85,B 0,C 180,E1 -5283.217,E2 -5283.217} C_VEL
LIN {X 0,Y 510.182,Z 392.583,A -85,B 0,C 180,E1 -5283.844,E2 -5283.844} C_VEL
LIN {X 0,Y 509.949,Z 399.89,A -85,B 0,C 180,E1 -5284.489,E2 -5284.489} C_VEL
LIN {X 0,Y 509.776,Z 407.014,A -85,B 0,C 180,E1 -5285.255,E2 -5285.255} C_VEL
LIN {X 0,Y 509.664,Z 412.736,A -85,B 0,C 180,E1 -5285.997,E2 -5285.997} C_VEL
LIN {X 0,Y 509.506,Z 418.22,A -85,B 0,C 180,E1 -5286.851,E2 -5286.851} C_VEL
LIN {X 0,Y 509.374,Z 423.379,A -85,B 0,C 180,E1 -5287.844,E2 -5287.844} C_VEL
LIN {X 0,Y 509.289,Z 427.946,A -85,B 0,C 180,E1 -5288.974,E2 -5288.974} C_VEL
LIN {X 0,Y 509.261,Z 430.456,A -85,B 0,C 180,E1 -5289.818,E2 -5289.818} C_VEL
LIN {X 0,Y 509.173,Z 432.333,A -85,B 0,C 180,E1 -5290.654,E2 -5290.654} C_VEL
LIN {X 0,Y 509.129,Z 433.639,A -85,B 0,C 180,E1 -5291.489,E2 -5291.489} C_VEL
LIN {X 0,Y 509.132,Z 434.405,A -85,B 0,C 180,E1 -5292.321,E2 -5292.321} C_VEL
LIN {X 0,Y 509.15,Z 434.65,A -85,B 0,C 180,E1 -5293.15,E2 -5293.15} C_VEL
LIN {X 0,Y 509.162,Z 434.313,A -85,B 0,C 180,E1 -5293.975,E2 -5293.975} C_VEL
LIN {X 0,Y 509.181,Z 433.085,A -85,B 0,C 180,E1 -5295.038,E2 -5295.038} C_VEL
LIN {X 0,Y 509.245,Z 429.979,A -85,B 0,C 180,E1 -5296.431,E2 -5296.431} C_VEL
LIN {X 0,Y 509.308,Z 425.891,A -85,B 0,C 180,E1 -5297.65,E2 -5297.65} C_VEL
LIN {X 0,Y 509.452,Z 420.356,A -85,B 0,C 180,E1 -5298.864,E2 -5298.864} C_VEL
LIN {X 0,Y 509.583,Z 414.272,A -85,B 0,C 180,E1 -5299.872,E2 -5299.872} C_VEL
LIN {X 0,Y 509.746,Z 408.311,A -85,B 0,C 180,E1 -5300.677,E2 -5300.677} C_VEL
LIN {X 0,Y 509.961,Z 401.05,A -85,B 0,C 180,E1 -5301.48,E2 -5301.48} C_VEL
LIN {X 0,Y 510.129,Z 393.471,A -85,B 0,C 180,E1 -5302.169,E2 -5302.169} C_VEL
LIN {X 0,Y 510.33,Z 385.101,A -85,B 0,C 180,E1 -5302.787,E2 -5302.787} C_VEL
LIN {X 0,Y 510.48,Z 376.752,A -85,B 0,C 180,E1 -5303.28,E2 -5303.28} C_VEL
LIN {X 0,Y 510.629,Z 366.886,A -85,B 0,C 180,E1 -5303.728,E2 -5303.728} C_VEL
LIN {X 0,Y 510.777,Z 354.704,A -85,B 0,C 180,E1 -5304.102,E2 -5304.102} C_VEL
LIN {X 0,Y 510.866,Z 334.256,A -85,B 0,C 180,E1 -5304.425,E2 -5304.425} C_VEL
LIN {X 0,Y 510.987,Z 284.138,A -85,B 0,C 180,E1 -5305.131,E2 -5305.131} C_VEL
LIN {X 0,Y 509.737,Z 276.352,A -85,B 0,C 180,E1 -5305.28,E2 -5305.28} C_VEL
LIN {X 0,Y 509.811,Z 260.967,A -85,B 0,C 180,E1 -5308.815,E2 -5308.815} C_VEL
LIN {X 0,Y 509.839,Z 256.789,A -85,B 0,C 180,E1 -5309.803,E2 -5309.803} C_VEL
LIN {X 0,Y 510.028,Z 256.767,A -85,B 0,C 180,E1 -5310.79,E2 -5310.79} C_VEL
LIN {X 0,Y 509.922,Z 256.782,A -85,B 0,C 180,E1 -5313.16,E2 -5313.16} C_VEL
LIN {X 0,Y 509.916,Z 256.775,A -85,B 0,C 180,E1 -5316.331,E2 -5316.331} C_VEL
LIN {X 0,Y 509.874,Z 256.782,A -85,B 0,C 180,E1 -5318.721,E2 -5318.721} C_VEL
LIN {X 0,Y 509.867,Z 256.783,A -85,B 0,C 180,E1 -5321.933,E2 -5321.933} C_VEL
LIN {X 0,Y 509.856,Z 256.79,A -85,B 0,C 180,E1 -5325.243,E2 -5325.243} C_VEL
LIN {X 0,Y 509.845,Z 256.785,A -85,B 0,C 180,E1 -5328,E2 -5328} C_VEL
LIN {X 0,Y 509.813,Z 256.791,A -85,B 0,C 180,E1 -5331.003,E2 -5331.003} C_VEL
LIN {X 0,Y 509.783,Z 256.798,A -85,B 0,C 180,E1 -5333.566,E2 -5333.566} C_VEL
LIN {X 0,Y 509.84,Z 256.784,A -85,B 0,C 180,E1 -5336.372,E2 -5336.372} C_VEL
LIN {X 0,Y 509.817,Z 256.788,A -85,B 0,C 180,E1 -5338.848,E2 -5338.848} C_VEL
LIN {X 0,Y 509.787,Z 256.799,A -85,B 0,C 180,E1 -5341.593,E2 -5341.593} C_VEL
LIN {X 0,Y 509.816,Z 256.787,A -85,B 0,C 180,E1 -5344.416,E2 -5344.416} C_VEL
LIN {X 0,Y 509.778,Z 256.798,A -85,B 0,C 180,E1 -5347.344,E2 -5347.344} C_VEL
LIN {X 0,Y 509.79,Z 256.791,A -85,B 0,C 180,E1 -5350.387,E2 -5350.387} C_VEL
LIN {X 0,Y 509.779,Z 256.794,A -85,B 0,C 180,E1 -5353.063,E2 -5353.063} C_VEL
LIN {X 0,Y 509.799,Z 256.796,A -85,B 0,C 180,E1 -5355.796,E2 -5355.796} C_VEL
LIN {X 0,Y 509.834,Z 256.785,A -85,B 0,C 180,E1 -5358.578,E2 -5358.578} C_VEL
LIN {X 0,Y 509.83,Z 256.794,A -85,B 0,C 180,E1 -5361.79,E2 -5361.79} C_VEL
LIN {X 0,Y 509.812,Z 256.788,A -85,B 0,C 180,E1 -5364.625,E2 -5364.625} C_VEL
LIN {X 0,Y 509.844,Z 256.789,A -85,B 0,C 180,E1 -5367.484,E2 -5367.484} C_VEL
LIN {X 0,Y 509.845,Z 256.786,A -85,B 0,C 180,E1 -5370.277,E2 -5370.277} C_VEL
LIN {X 0,Y 509.84,Z 256.785,A -85,B 0,C 180,E1 -5372.946,E2 -5372.946} C_VEL
LIN {X 0,Y 509.835,Z 256.791,A -85,B 0,C 180,E1 -5375.576,E2 -5375.576} C_VEL
LIN {X 0,Y 509.813,Z 256.793,A -85,B 0,C 180,E1 -5378.152,E2 -5378.152} C_VEL
LIN {X 0,Y 509.848,Z 256.784,A -85,B 0,C 180,E1 -5380.684,E2 -5380.684} C_VEL
LIN {X 0,Y 509.85,Z 256.852,A -85,B 0,C 180,E1 -5383.228,E2 -5383.228} C_VEL
LIN {X 0,Y 509.79,Z 266.99,A -85,B 0,C 180,E1 -5385.635,E2 -5385.635} C_VEL
LIN {X 0,Y 509.667,Z 276.33,A -85,B 0,C 180,E1 -5387.843,E2 -5387.843} C_VEL
LIN {X 0,Y 511.058,Z 285.56,A -85,B 0,C 180,E1 -5388.02,E2 -5388.02} C_VEL
LIN {X 0,Y 510.707,Z 353.129,A -85,B 0,C 180,E1 -5389.046,E2 -5389.046} C_VEL
LIN {X 0,Y 510.577,Z 363.005,A -85,B 0,C 180,E1 -5389.319,E2 -5389.319} C_VEL
LIN {X 0,Y 510.434,Z 372.389,A -85,B 0,C 180,E1 -5389.692,E2 -5389.692} C_VEL
LIN {X 0,Y 510.282,Z 381.814,A -85,B 0,C 180,E1 -5390.19,E2 -5390.19} C_VEL
LIN {X 0,Y 510.118,Z 391.932,A -85,B 0,C 180,E1 -5390.887,E2 -5390.887} C_VEL
LIN {X 0,Y 509.869,Z 400.804,A -85,B 0,C 180,E1 -5391.681,E2 -5391.681} C_VEL
LIN {X 0,Y 509.705,Z 408.022,A -85,B 0,C 180,E1 -5392.476,E2 -5392.476} C_VEL
LIN {X 0,Y 509.612,Z 413.425,A -85,B 0,C 180,E1 -5393.192,E2 -5393.192} C_VEL
LIN {X 0,Y 509.526,Z 418.912,A -85,B 0,C 180,E1 -5394.065,E2 -5394.065} C_VEL
LIN {X 0,Y 509.345,Z 423.016,A -85,B 0,C 180,E1 -5394.857,E2 -5394.857} C_VEL
LIN {X 0,Y 509.373,Z 426.395,A -85,B 0,C 180,E1 -5395.651,E2 -5395.651} C_VEL
LIN {X 0,Y 509.314,Z 430.275,A -85,B 0,C 180,E1 -5396.839,E2 -5396.839} C_VEL
LIN {X 0,Y 509.199,Z 432.12,A -85,B 0,C 180,E1 -5397.63,E2 -5397.63} C_VEL
LIN {X 0,Y 509.114,Z 433.45,A -85,B 0,C 180,E1 -5398.421,E2 -5398.421} C_VEL
LIN {X 0,Y 509.085,Z 434.288,A -85,B 0,C 180,E1 -5399.212,E2 -5399.212} C_VEL
LIN {X 0,Y 509.084,Z 434.605,A -85,B 0,C 180,E1 -5400.003,E2 -5400.003} C_VEL
LIN {X 0,Y 509.086,Z 434.345,A -85,B 0,C 180,E1 -5400.794,E2 -5400.794} C_VEL
LIN {X 0,Y 509.115,Z 433.595,A -85,B 0,C 180,E1 -5401.585,E2 -5401.585} C_VEL
LIN {X 0,Y 509.201,Z 432.352,A -85,B 0,C 180,E1 -5402.376,E2 -5402.376} C_VEL
LIN {X 0,Y 509.341,Z 429.476,A -85,B 0,C 180,E1 -5403.562,E2 -5403.562} C_VEL
LIN {X 0,Y 509.394,Z 425.331,A -85,B 0,C 180,E1 -5404.751,E2 -5404.751} C_VEL
LIN {X 0,Y 509.519,Z 419.523,A -85,B 0,C 180,E1 -5405.94,E2 -5405.94} C_VEL
LIN {X 0,Y 509.571,Z 414.447,A -85,B 0,C 180,E1 -5406.77,E2 -5406.77} C_VEL
LIN {X 0,Y 509.705,Z 408.855,A -85,B 0,C 180,E1 -5407.529,E2 -5407.529} C_VEL
LIN {X 0,Y 509.844,Z 401.763,A -85,B 0,C 180,E1 -5408.324,E2 -5408.324} C_VEL
LIN {X 0,Y 510.053,Z 394.197,A -85,B 0,C 180,E1 -5409.02,E2 -5409.02} C_VEL
LIN {X 0,Y 510.285,Z 384.846,A -85,B 0,C 180,E1 -5409.715,E2 -5409.715} C_VEL
LIN {X 0,Y 510.447,Z 374.157,A -85,B 0,C 180,E1 -5410.313,E2 -5410.313} C_VEL
LIN {X 0,Y 510.549,Z 364.493,A -85,B 0,C 180,E1 -5410.712,E2 -5410.712} C_VEL
LIN {X 0,Y 510.63,Z 355.102,A -85,B 0,C 180,E1 -5410.986,E2 -5410.986} C_VEL
LIN {X 0,Y 510.798,Z 341.771,A -85,B 0,C 180,E1 -5411.22,E2 -5411.22} C_VEL
LIN {X 0,Y 510.938,Z 284.127,A -85,B 0,C 180,E1 -5412.092,E2 -5412.092} C_VEL
LIN {X 0,Y 509.722,Z 276.94,A -85,B 0,C 180,E1 -5412.24,E2 -5412.24} C_VEL
LIN {X 0,Y 509.819,Z 262.468,A -85,B 0,C 180,E1 -5415.555,E2 -5415.555} C_VEL
LIN {X 0,Y 509.869,Z 256.789,A -85,B 0,C 180,E1 -5416.879,E2 -5416.879} C_VEL
LIN {X 0,Y 509.924,Z 256.784,A -85,B 0,C 180,E1 -5420.157,E2 -5420.157} C_VEL
LIN {X 0,Y 509.827,Z 256.788,A -85,B 0,C 180,E1 -5423.565,E2 -5423.565} C_VEL
LIN {X 0,Y 509.845,Z 256.792,A -85,B 0,C 180,E1 -5426.363,E2 -5426.363} C_VEL
LIN {X 0,Y 509.858,Z 256.786,A -85,B 0,C 180,E1 -5428.847,E2 -5428.847} C_VEL
LIN {X 0,Y 509.826,Z 256.788,A -85,B 0,C 180,E1 -5431.591,E2 -5431.591} C_VEL
LIN {X 0,Y 509.845,Z 256.793,A -85,B 0,C 180,E1 -5434.416,E2 -5434.416} C_VEL
LIN {X 0,Y 509.816,Z 256.789,A -85,B 0,C 180,E1 -5437.342,E2 -5437.342} C_VEL
LIN {X 0,Y 509.826,Z 256.795,A -85,B 0,C 180,E1 -5440.385,E2 -5440.385} C_VEL
LIN {X 0,Y 509.812,Z 256.79,A -85,B 0,C 180,E1 -5443.06,E2 -5443.06} C_VEL
LIN {X 0,Y 509.83,Z 256.786,A -85,B 0,C 180,E1 -5445.794,E2 -5445.794} C_VEL
LIN {X 0,Y 509.853,Z 256.791,A -85,B 0,C 180,E1 -5448.574,E2 -5448.574} C_VEL
LIN {X 0,Y 509.856,Z 256.783,A -85,B 0,C 180,E1 -5451.787,E2 -5451.787} C_VEL
LIN {X 0,Y 509.833,Z 256.793,A -85,B 0,C 180,E1 -5454.622,E2 -5454.622} C_VEL
LIN {X 0,Y 509.866,Z 256.783,A -85,B 0,C 180,E1 -5457.481,E2 -5457.481} C_VEL
LIN {X 0,Y 509.865,Z 256.786,A -85,B 0,C 180,E1 -5460.274,E2 -5460.274} C_VEL
LIN {X 0,Y 509.888,Z 256.786,A -85,B 0,C 180,E1 -5462.944,E2 -5462.944} C_VEL
LIN {X 0,Y 509.895,Z 256.785,A -85,B 0,C 180,E1 -5466.386,E2 -5466.386} C_VEL
LIN {X 0,Y 510.855,Z 262.828,A -85,B 0,C 180,E1 -5467.557,E2 -5467.557} C_VEL
LIN {X 0,Y 510.611,Z 275.76,A -85,B 0,C 180,E1 -5469.873,E2 -5469.873} C_VEL
LIN {X 0,Y 510.232,Z 292.154,A -85,B 0,C 180,E1 -5472.774,E2 -5472.774} C_VEL
LIN {X 0,Y 509.906,Z 309.665,A -85,B 0,C 180,E1 -5475.839,E2 -5475.839} C_VEL
LIN {X 0,Y 509.701,Z 320.616,A -85,B 0,C 180,E1 -5477.741,E2 -5477.741} C_VEL
LIN {X 0,Y 511.056,Z 333.176,A -85,B 0,C 180,E1 -5477.957,E2 -5477.957} C_VEL
LIN {X 0,Y 510.767,Z 398.388,A -85,B 0,C 180,E1 -5478.893,E2 -5478.893} C_VEL
LIN {X 0,Y 510.55,Z 408.117,A -85,B 0,C 180,E1 -5479.139,E2 -5479.139} C_VEL
LIN {X 0,Y 510.374,Z 419.739,A -85,B 0,C 180,E1 -5479.587,E2 -5479.587} C_VEL
LIN {X 0,Y 510.171,Z 430.416,A -85,B 0,C 180,E1 -5480.184,E2 -5480.184} C_VEL
LIN {X 0,Y 509.987,Z 438.772,A -85,B 0,C 180,E1 -5480.781,E2 -5480.781} C_VEL
LIN {X 0,Y 509.803,Z 446.68,A -85,B 0,C 180,E1 -5481.477,E2 -5481.477} C_VEL
LIN {X 0,Y 509.585,Z 454.072,A -85,B 0,C 180,E1 -5482.272,E2 -5482.272} C_VEL
LIN {X 0,Y 509.492,Z 460.582,A -85,B 0,C 180,E1 -5483.127,E2 -5483.127} C_VEL
LIN {X 0,Y 509.37,Z 467.47,A -85,B 0,C 180,E1 -5484.259,E2 -5484.259} C_VEL
LIN {X 0,Y 509.225,Z 472.105,A -85,B 0,C 180,E1 -5485.25,E2 -5485.25} C_VEL
LIN {X 0,Y 509.259,Z 475.121,A -85,B 0,C 180,E1 -5486.043,E2 -5486.043} C_VEL
LIN {X 0,Y 509.213,Z 477.456,A -85,B 0,C 180,E1 -5486.835,E2 -5486.835} C_VEL
LIN {X 0,Y 509.193,Z 479.214,A -85,B 0,C 180,E1 -5487.627,E2 -5487.627} C_VEL
LIN {X 0,Y 509.112,Z 480.47,A -85,B 0,C 180,E1 -5488.418,E2 -5488.418} C_VEL
LIN {X 0,Y 509.077,Z 481.252,A -85,B 0,C 180,E1 -5489.209,E2 -5489.209} C_VEL
LIN {X 0,Y 509.075,Z 481.546,A -85,B 0,C 180,E1 -5490,E2 -5490} C_VEL
LIN {X 0,Y 509.077,Z 481.247,A -85,B 0,C 180,E1 -5490.791,E2 -5490.791} C_VEL
LIN {X 0,Y 509.112,Z 480.461,A -85,B 0,C 180,E1 -5491.582,E2 -5491.582} C_VEL
LIN {X 0,Y 509.193,Z 479.201,A -85,B 0,C 180,E1 -5492.373,E2 -5492.373} C_VEL
LIN {X 0,Y 509.244,Z 476.278,A -85,B 0,C 180,E1 -5493.56,E2 -5493.56} C_VEL
LIN {X 0,Y 509.235,Z 473.612,A -85,B 0,C 180,E1 -5494.353,E2 -5494.353} C_VEL
LIN {X 0,Y 509.336,Z 468.401,A -85,B 0,C 180,E1 -5495.543,E2 -5495.543} C_VEL
LIN {X 0,Y 509.456,Z 462.038,A -85,B 0,C 180,E1 -5496.659,E2 -5496.659} C_VEL
LIN {X 0,Y 509.584,Z 454.032,A -85,B 0,C 180,E1 -5497.728,E2 -5497.728} C_VEL
LIN {X 0,Y 509.801,Z 446.639,A -85,B 0,C 180,E1 -5498.522,E2 -5498.522} C_VEL
LIN {X 0,Y 509.976,Z 438.723,A -85,B 0,C 180,E1 -5499.219,E2 -5499.219} C_VEL
LIN {X 0,Y 510.171,Z 430.36,A -85,B 0,C 180,E1 -5499.815,E2 -5499.815} C_VEL
LIN {X 0,Y 510.374,Z 419.681,A -85,B 0,C 180,E1 -5500.412,E2 -5500.412} C_VEL
LIN {X 0,Y 510.57,Z 408.056,A -85,B 0,C 180,E1 -5500.86,E2 -5500.86} C_VEL
LIN {X 0,Y 510.768,Z 398.322,A -85,B 0,C 180,E1 -5501.106,E2 -5501.106} C_VEL
LIN {X 0,Y 510.867,Z 330.332,A -85,B 0,C 180,E1 -5502.086,E2 -5502.086} C_VEL
LIN {X 0,Y 509.698,Z 320.44,A -85,B 0,C 180,E1 -5502.27,E2 -5502.27} C_VEL
LIN {X 0,Y 509.941,Z 303.606,A -85,B 0,C 180,E1 -5505.18,E2 -5505.18} C_VEL
LIN {X 0,Y 510.373,Z 284.788,A -85,B 0,C 180,E1 -5508.464,E2 -5508.464} C_VEL
LIN {X 0,Y 510.75,Z 267.065,A -85,B 0,C 180,E1 -5511.597,E2 -5511.597} C_VEL
LIN {X 0,Y 510.627,Z 261.148,A -85,B 0,C 180,E1 -5512.667,E2 -5512.667} C_VEL
LIN {X 0,Y 509.88,Z 256.788,A -85,B 0,C 180,E1 -5513.507,E2 -5513.507} C_VEL
LIN {X 0,Y 509.915,Z 256.778,A -85,B 0,C 180,E1 -5516.378,E2 -5516.378} C_VEL
LIN {X 0,Y 509.877,Z 256.784,A -85,B 0,C 180,E1 -5518.844,E2 -5518.844} C_VEL
LIN {X 0,Y 509.824,Z 256.79,A -85,B 0,C 180,E1 -5521.59,E2 -5521.59} C_VEL
LIN {X 0,Y 509.843,Z 256.786,A -85,B 0,C 180,E1 -5524.414,E2 -5524.414} C_VEL
LIN {X 0,Y 509.821,Z 256.794,A -85,B 0,C 180,E1 -5527.34,E2 -5527.34} C_VEL
LIN {X 0,Y 509.844,Z 256.785,A -85,B 0,C 180,E1 -5530.382,E2 -5530.382} C_VEL
LIN {X 0,Y 509.813,Z 256.792,A -85,B 0,C 180,E1 -5533.059,E2 -5533.059} C_VEL
LIN {X 0,Y 509.829,Z 256.791,A -85,B 0,C 180,E1 -5535.792,E2 -5535.792} C_VEL
LIN {X 0,Y 509.861,Z 256.782,A -85,B 0,C 180,E1 -5538.573,E2 -5538.573} C_VEL
LIN {X 0,Y 509.856,Z 256.789,A -85,B 0,C 180,E1 -5541.786,E2 -5541.786} C_VEL
LIN {X 0,Y 509.835,Z 256.783,A -85,B 0,C 180,E1 -5544.621,E2 -5544.621} C_VEL
LIN {X 0,Y 509.866,Z 256.788,A -85,B 0,C 180,E1 -5547.48,E2 -5547.48} C_VEL
LIN {X 0,Y 509.864,Z 256.783,A -85,B 0,C 180,E1 -5550.273,E2 -5550.273} C_VEL
LIN {X 0,Y 509.89,Z 256.784,A -85,B 0,C 180,E1 -5553.626,E2 -5553.626} C_VEL
LIN {X 0,Y 509.827,Z 256.787,A -85,B 0,C 180,E1 -5556.435,E2 -5556.435} C_VEL
LIN {X 0,Y 509.92,Z 256.781,A -85,B 0,C 180,E1 -5559.843,E2 -5559.843} C_VEL
LIN {X 0,Y 509.873,Z 256.779,A -85,B 0,C 180,E1 -5563.172,E2 -5563.172} C_VEL
LIN {X 0,Y 509.866,Z 256.784,A -85,B 0,C 180,E1 -5565.632,E2 -5565.632} C_VEL
LIN {X 0,Y 509.916,Z 256.77,A -85,B 0,C 180,E1 -5568.872,E2 -5568.872} C_VEL
LIN {X 0,Y 509.954,Z 256.776,A -85,B 0,C 180,E1 -5572.076,E2 -5572.076} C_VEL
LIN {X 0,Y 509.98,Z 256.766,A -85,B 0,C 180,E1 -5574.462,E2 -5574.462} C_VEL
LIN {X 0,Y 510.052,Z 256.76,A -85,B 0,C 180,E1 -5577.628,E2 -5577.628} C_VEL
LIN {X 0,Y 510.057,Z 256.761,A -85,B 0,C 180,E1 -5579.997,E2 -5579.997} C_VEL
LIN {X 0,Y 510.05,Z 256.763,A -85,B 0,C 180,E1 -5582.366,E2 -5582.366} C_VEL
LIN {X 0,Y 509.968,Z 256.765,A -85,B 0,C 180,E1 -5585.533,E2 -5585.533} C_VEL
LIN {X 0,Y 509.907,Z 256.777,A -85,B 0,C 180,E1 -5588.717,E2 -5588.717} C_VEL
LIN {X 0,Y 509.9,Z 256.779,A -85,B 0,C 180,E1 -5591.929,E2 -5591.929} C_VEL
LIN {X 0,Y 509.888,Z 256.776,A -85,B 0,C 180,E1 -5595.239,E2 -5595.239} C_VEL
LIN {X 0,Y 509.853,Z 256.789,A -85,B 0,C 180,E1 -5598.481,E2 -5598.481} C_VEL
LIN {X 0,Y 509.84,Z 256.785,A -85,B 0,C 180,E1 -5600.999,E2 -5600.999} C_VEL
LIN {X 0,Y 509.852,Z 256.789,A -85,B 0,C 180,E1 -5604.423,E2 -5604.423} C_VEL
LIN {X 0,Y 509.872,Z 256.782,A -85,B 0,C 180,E1 -5607.052,E2 -5607.052} C_VEL
LIN {X 0,Y 509.842,Z 256.785,A -85,B 0,C 180,E1 -5609.748,E2 -5609.748} C_VEL
LIN {X 0,Y 509.857,Z 256.788,A -85,B 0,C 180,E1 -5612.771,E2 -5612.771} C_VEL
LIN {X 0,Y 509.82,Z 256.783,A -85,B 0,C 180,E1 -5615.578,E2 -5615.578} C_VEL
LIN {X 0,Y 509.829,Z 256.791,A -85,B 0,C 180,E1 -5618.335,E2 -5618.335} C_VEL
LIN {X 0,Y 509.842,Z 256.785,A -85,B 0,C 180,E1 -5621.422,E2 -5621.422} C_VEL
LIN {X 0,Y 509.832,Z 256.792,A -85,B 0,C 180,E1 -5624.665,E2 -5624.665} C_VEL
LIN {X 0,Y 509.86,Z 256.784,A -85,B 0,C 180,E1 -5628.097,E2 -5628.097} C_VEL
LIN {X 0,Y 509.849,Z 256.792,A -85,B 0,C 180,E1 -5630.648,E2 -5630.648} C_VEL
LIN {X 0,Y 509.805,Z 256.792,A -85,B 0,C 180,E1 -5633.713,E2 -5633.713} C_VEL
LIN {X 0,Y 509.122,Z 256.878,A -85,B 0,C 180,E1 -5634.153,E2 -5634.153} C_VEL
LIN {X 0,Y 506.285,Z 257.236,A -85,B 0,C 180,E1 -5634.841,E2 -5634.841} C_VEL
LIN {X 0,Y 503.439,Z 257.587,A -85,B 0,C 180,E1 -5635.537,E2 -5635.537} C_VEL
LIN {X 0,Y 502.759,Z 257.671,A -85,B 0,C 180,E1 -5635.985,E2 -5635.985} C_VEL
LIN {X 0,Y 502.716,Z 257.718,A -85,B 0,C 180,E1 -5636.481,E2 -5636.481} C_VEL
LIN {X 0,Y 502.655,Z 269.511,A -85,B 0,C 180,E1 -5639.081,E2 -5639.081} C_VEL
LIN {X 0,Y 502.642,Z 276.429,A -85,B 0,C 180,E1 -5640.622,E2 -5640.622} C_VEL
LIN {X 0,Y 504.228,Z 286.789,A -85,B 0,C 180,E1 -5640.826,E2 -5640.826} C_VEL
LIN {X 0,Y 503.869,Z 352.833,A -85,B 0,C 180,E1 -5641.79,E2 -5641.79} C_VEL
LIN {X 0,Y 503.721,Z 363.645,A -85,B 0,C 180,E1 -5642.078,E2 -5642.078} C_VEL
LIN {X 0,Y 503.563,Z 375.464,A -85,B 0,C 180,E1 -5642.577,E2 -5642.577} C_VEL
LIN {X 0,Y 503.394,Z 384.546,A -85,B 0,C 180,E1 -5643.104,E2 -5643.104} C_VEL
LIN {X 0,Y 503.206,Z 392.437,A -85,B 0,C 180,E1 -5643.677,E2 -5643.677} C_VEL
LIN {X 0,Y 502.94,Z 399.82,A -85,B 0,C 180,E1 -5644.33,E2 -5644.33} C_VEL
LIN {X 0,Y 502.786,Z 406.003,A -85,B 0,C 180,E1 -5644.986,E2 -5644.986} C_VEL
LIN {X 0,Y 502.631,Z 412.794,A -85,B 0,C 180,E1 -5645.859,E2 -5645.859} C_VEL
LIN {X 0,Y 502.459,Z 418.323,A -85,B 0,C 180,E1 -5646.726,E2 -5646.726} C_VEL
LIN {X 0,Y 502.378,Z 421.965,A -85,B 0,C 180,E1 -5647.402,E2 -5647.402} C_VEL
LIN {X 0,Y 502.235,Z 427.33,A -85,B 0,C 180,E1 -5648.665,E2 -5648.665} C_VEL
LIN {X 0,Y 502.206,Z 430.411,A -85,B 0,C 180,E1 -5649.642,E2 -5649.642} C_VEL
LIN {X 0,Y 502.109,Z 432.162,A -85,B 0,C 180,E1 -5650.371,E2 -5650.371} C_VEL
LIN {X 0,Y 502.063,Z 433.671,A -85,B 0,C 180,E1 -5651.219,E2 -5651.219} C_VEL
LIN {X 0,Y 502.042,Z 434.667,A -85,B 0,C 180,E1 -5652.146,E2 -5652.146} C_VEL
LIN {X 0,Y 502.059,Z 434.964,A -85,B 0,C 180,E1 -5652.905,E2 -5652.905} C_VEL
LIN {X 0,Y 502.069,Z 434.739,A -85,B 0,C 180,E1 -5653.742,E2 -5653.742} C_VEL
LIN {X 0,Y 502.097,Z 433.553,A -85,B 0,C 180,E1 -5654.957,E2 -5654.957} C_VEL
LIN {X 0,Y 502.139,Z 430.997,A -85,B 0,C 180,E1 -5656.235,E2 -5656.235} C_VEL
LIN {X 0,Y 502.213,Z 428.623,A -85,B 0,C 180,E1 -5657.062,E2 -5657.062} C_VEL
LIN {X 0,Y 502.318,Z 423.661,A -85,B 0,C 180,E1 -5658.321,E2 -5658.321} C_VEL
LIN {X 0,Y 502.458,Z 418.541,A -85,B 0,C 180,E1 -5659.32,E2 -5659.32} C_VEL
LIN {X 0,Y 502.559,Z 413.414,A -85,B 0,C 180,E1 -5660.136,E2 -5660.136} C_VEL
LIN {X 0,Y 502.7,Z 407.233,A -85,B 0,C 180,E1 -5660.951,E2 -5660.951} C_VEL
LIN {X 0,Y 502.971,Z 400.698,A -85,B 0,C 180,E1 -5661.665,E2 -5661.665} C_VEL
LIN {X 0,Y 503.135,Z 393.127,A -85,B 0,C 180,E1 -5662.351,E2 -5662.351} C_VEL
LIN {X 0,Y 503.342,Z 386.024,A -85,B 0,C 180,E1 -5662.882,E2 -5662.882} C_VEL
LIN {X 0,Y 503.493,Z 377.717,A -85,B 0,C 180,E1 -5663.387,E2 -5663.387} C_VEL
LIN {X 0,Y 503.65,Z 369.232,A -85,B 0,C 180,E1 -5663.792,E2 -5663.792} C_VEL
LIN {X 0,Y 503.783,Z 359.149,A -85,B 0,C 180,E1 -5664.145,E2 -5664.145} C_VEL
LIN {X 0,Y 503.898,Z 347.603,A -85,B 0,C 180,E1 -5664.397,E2 -5664.397} C_VEL
LIN {X 0,Y 504.085,Z 285.051,A -85,B 0,C 180,E1 -5665.289,E2 -5665.289} C_VEL
LIN {X 0,Y 502.711,Z 276.533,A -85,B 0,C 180,E1 -5665.465,E2 -5665.465} C_VEL
LIN {X 0,Y 502.784,Z 262.099,A -85,B 0,C 180,E1 -5668.799,E2 -5668.799} C_VEL
LIN {X 0,Y 502.812,Z 257.664,A -85,B 0,C 180,E1 -5669.85,E2 -5669.85} C_VEL
LIN {X 0,Y 502.998,Z 257.643,A -85,B 0,C 180,E1 -5670.801,E2 -5670.801} C_VEL
LIN {X 0,Y 502.866,Z 257.662,A -85,B 0,C 180,E1 -5673.205,E2 -5673.205} C_VEL
LIN {X 0,Y 502.869,Z 257.653,A -85,B 0,C 180,E1 -5676.42,E2 -5676.42} C_VEL
LIN {X 0,Y 502.834,Z 257.66,A -85,B 0,C 180,E1 -5678.844,E2 -5678.844} C_VEL
LIN {X 0,Y 502.808,Z 257.661,A -85,B 0,C 180,E1 -5682.103,E2 -5682.103} C_VEL
LIN {X 0,Y 502.811,Z 257.668,A -85,B 0,C 180,E1 -5685.401,E2 -5685.401} C_VEL
LIN {X 0,Y 502.804,Z 257.661,A -85,B 0,C 180,E1 -5688.122,E2 -5688.122} C_VEL
LIN {X 0,Y 502.793,Z 257.662,A -85,B 0,C 180,E1 -5690.538,E2 -5690.538} C_VEL
LIN {X 0,Y 502.751,Z 257.671,A -85,B 0,C 180,E1 -5693.043,E2 -5693.043} C_VEL
LIN {X 0,Y 502.81,Z 257.66,A -85,B 0,C 180,E1 -5696.558,E2 -5696.558} C_VEL
LIN {X 0,Y 502.782,Z 257.666,A -85,B 0,C 180,E1 -5699.937,E2 -5699.937} C_VEL
LIN {X 0,Y 502.801,Z 257.664,A -85,B 0,C 180,E1 -5703.034,E2 -5703.034} C_VEL
LIN {X 0,Y 502.738,Z 257.672,A -85,B 0,C 180,E1 -5705.954,E2 -5705.954} C_VEL
LIN {X 0,Y 502.765,Z 257.667,A -85,B 0,C 180,E1 -5708.98,E2 -5708.98} C_VEL
LIN {X 0,Y 502.778,Z 257.666,A -85,B 0,C 180,E1 -5712.202,E2 -5712.202} C_VEL
LIN {X 0,Y 502.762,Z 257.673,A -85,B 0,C 180,E1 -5715.473,E2 -5715.473} C_VEL
LIN {X 0,Y 502.799,Z 257.663,A -85,B 0,C 180,E1 -5718.937,E2 -5718.937} C_VEL
LIN {X 0,Y 502.772,Z 257.669,A -85,B 0,C 180,E1 -5722.049,E2 -5722.049} C_VEL
LIN {X 0,Y 502.778,Z 257.666,A -85,B 0,C 180,E1 -5725.037,E2 -5725.037} C_VEL
LIN {X 0,Y 502.767,Z 257.672,A -85,B 0,C 180,E1 -5727.919,E2 -5727.919} C_VEL
LIN {X 0,Y 502.799,Z 257.662,A -85,B 0,C 180,E1 -5730.715,E2 -5730.715} C_VEL
LIN {X 0,Y 502.789,Z 257.667,A -85,B 0,C 180,E1 -5733.457,E2 -5733.457} C_VEL
LIN {X 0,Y 502.763,Z 257.671,A -85,B 0,C 180,E1 -5736.089,E2 -5736.089} C_VEL
LIN {X 0,Y 502.775,Z 257.665,A -85,B 0,C 180,E1 -5738.692,E2 -5738.692} C_VEL
LIN {X 0,Y 502.805,Z 257.663,A -85,B 0,C 180,E1 -5741.251,E2 -5741.251} C_VEL
LIN {X 0,Y 502.794,Z 257.688,A -85,B 0,C 180,E1 -5743.195,E2 -5743.195} C_VEL
LIN {X 0,Y 502.728,Z 268.837,A -85,B 0,C 180,E1 -5745.842,E2 -5745.842} C_VEL
LIN {X 0,Y 502.635,Z 276.56,A -85,B 0,C 180,E1 -5747.676,E2 -5747.676} C_VEL
LIN {X 0,Y 504.104,Z 286.948,A -85,B 0,C 180,E1 -5747.876,E2 -5747.876} C_VEL
LIN {X 0,Y 503.745,Z 352.805,A -85,B 0,C 180,E1 -5748.892,E2 -5748.892} C_VEL
LIN {X 0,Y 503.608,Z 362.85,A -85,B 0,C 180,E1 -5749.169,E2 -5749.169} C_VEL
LIN {X 0,Y 503.437,Z 372.332,A -85,B 0,C 180,E1 -5749.547,E2 -5749.547} C_VEL
LIN {X 0,Y 503.304,Z 380.09,A -85,B 0,C 180,E1 -5749.951,E2 -5749.951} C_VEL
LIN {X 0,Y 503.159,Z 389.32,A -85,B 0,C 180,E1 -5750.557,E2 -5750.557} C_VEL
LIN {X 0,Y 502.9,Z 398.981,A -85,B 0,C 180,E1 -5751.363,E2 -5751.363} C_VEL
LIN {X 0,Y 502.702,Z 406.551,A -85,B 0,C 180,E1 -5752.169,E2 -5752.169} C_VEL
LIN {X 0,Y 502.559,Z 412.761,A -85,B 0,C 180,E1 -5752.969,E2 -5752.969} C_VEL
LIN {X 0,Y 502.545,Z 417.994,A -85,B 0,C 180,E1 -5753.781,E2 -5753.781} C_VEL
LIN {X 0,Y 502.271,Z 423.264,A -85,B 0,C 180,E1 -5754.784,E2 -5754.784} C_VEL
LIN {X 0,Y 502.313,Z 426.658,A -85,B 0,C 180,E1 -5755.589,E2 -5755.589} C_VEL
LIN {X 0,Y 502.23,Z 430.562,A -85,B 0,C 180,E1 -5756.794,E2 -5756.794} C_VEL
LIN {X 0,Y 502.134,Z 432.415,A -85,B 0,C 180,E1 -5757.596,E2 -5757.596} C_VEL
LIN {X 0,Y 502.038,Z 433.753,A -85,B 0,C 180,E1 -5758.398,E2 -5758.398} C_VEL
LIN {X 0,Y 502.001,Z 434.598,A -85,B 0,C 180,E1 -5759.2,E2 -5759.2} C_VEL
LIN {X 0,Y 501.998,Z 434.919,A -85,B 0,C 180,E1 -5760.003,E2 -5760.003} C_VEL
LIN {X 0,Y 502.002,Z 434.66,A -85,B 0,C 180,E1 -5760.805,E2 -5760.805} C_VEL
LIN {X 0,Y 502.039,Z 433.907,A -85,B 0,C 180,E1 -5761.607,E2 -5761.607} C_VEL
LIN {X 0,Y 502.136,Z 432.659,A -85,B 0,C 180,E1 -5762.409,E2 -5762.409} C_VEL
LIN {X 0,Y 502.253,Z 429.771,A -85,B 0,C 180,E1 -5763.613,E2 -5763.613} C_VEL
LIN {X 0,Y 502.321,Z 425.608,A -85,B 0,C 180,E1 -5764.818,E2 -5764.818} C_VEL
LIN {X 0,Y 502.411,Z 420.908,A -85,B 0,C 180,E1 -5765.823,E2 -5765.823} C_VEL
LIN {X 0,Y 502.511,Z 415.207,A -85,B 0,C 180,E1 -5766.786,E2 -5766.786} C_VEL
LIN {X 0,Y 502.665,Z 409.045,A -85,B 0,C 180,E1 -5767.635,E2 -5767.635} C_VEL
LIN {X 0,Y 502.84,Z 401.927,A -85,B 0,C 180,E1 -5768.441,E2 -5768.441} C_VEL
LIN {X 0,Y 503.05,Z 394.332,A -85,B 0,C 180,E1 -5769.146,E2 -5769.146} C_VEL
LIN {X 0,Y 503.294,Z 384.939,A -85,B 0,C 180,E1 -5769.852,E2 -5769.852} C_VEL
LIN {X 0,Y 503.447,Z 374.141,A -85,B 0,C 180,E1 -5770.458,E2 -5770.458} C_VEL
LIN {X 0,Y 503.571,Z 364.387,A -85,B 0,C 180,E1 -5770.862,E2 -5770.862} C_VEL
LIN {X 0,Y 503.683,Z 354.835,A -85,B 0,C 180,E1 -5771.14,E2 -5771.14} C_VEL
LIN {X 0,Y 503.871,Z 336.012,A -85,B 0,C 180,E1 -5771.456,E2 -5771.456} C_VEL
LIN {X 0,Y 504.08,Z 285.356,A -85,B 0,C 180,E1 -5772.242,E2 -5772.242} C_VEL
LIN {X 0,Y 502.675,Z 277.16,A -85,B 0,C 180,E1 -5772.415,E2 -5772.415} C_VEL
LIN {X 0,Y 502.795,Z 264.242,A -85,B 0,C 180,E1 -5775.403,E2 -5775.403} C_VEL
LIN {X 0,Y 502.857,Z 257.663,A -85,B 0,C 180,E1 -5776.913,E2 -5776.913} C_VEL
LIN {X 0,Y 502.828,Z 257.665,A -85,B 0,C 180,E1 -5779.602,E2 -5779.602} C_VEL
LIN {X 0,Y 502.811,Z 257.665,A -85,B 0,C 180,E1 -5782.704,E2 -5782.704} C_VEL
LIN {X 0,Y 502.788,Z 257.667,A -85,B 0,C 180,E1 -5785.68,E2 -5785.68} C_VEL
LIN {X 0,Y 502.804,Z 257.669,A -85,B 0,C 180,E1 -5788.377,E2 -5788.377} C_VEL
LIN {X 0,Y 502.802,Z 257.663,A -85,B 0,C 180,E1 -5791.145,E2 -5791.145} C_VEL
LIN {X 0,Y 502.796,Z 257.666,A -85,B 0,C 180,E1 -5793.996,E2 -5793.996} C_VEL
LIN {X 0,Y 502.772,Z 257.667,A -85,B 0,C 180,E1 -5797.176,E2 -5797.176} C_VEL
LIN {X 0,Y 502.781,Z 257.667,A -85,B 0,C 180,E1 -5800.017,E2 -5800.017} C_VEL
LIN {X 0,Y 502.812,Z 257.665,A -85,B 0,C 180,E1 -5802.2,E2 -5802.2} C_VEL
LIN {X 0,Y 502.793,Z 257.662,A -85,B 0,C 180,E1 -5805.471,E2 -5805.471} C_VEL
LIN {X 0,Y 502.803,Z 257.662,A -85,B 0,C 180,E1 -5807.861,E2 -5807.861} C_VEL
LIN {X 0,Y 502.803,Z 257.665,A -85,B 0,C 180,E1 -5811.024,E2 -5811.024} C_VEL
LIN {X 0,Y 502.778,Z 257.666,A -85,B 0,C 180,E1 -5814.17,E2 -5814.17} C_VEL
LIN {X 0,Y 502.81,Z 257.666,A -85,B 0,C 180,E1 -5816.999,E2 -5816.999} C_VEL
LIN {X 0,Y 502.821,Z 257.661,A -85,B 0,C 180,E1 -5820.065,E2 -5820.065} C_VEL
LIN {X 0,Y 502.834,Z 257.665,A -85,B 0,C 180,E1 -5822.533,E2 -5822.533} C_VEL
LIN {X 0,Y 502.792,Z 257.669,A -85,B 0,C 180,E1 -5825.309,E2 -5825.309} C_VEL
LIN {X 0,Y 502.859,Z 257.69,A -85,B 0,C 180,E1 -5826.308,E2 -5826.308} C_VEL
LIN {X 0,Y 503.906,Z 264.85,A -85,B 0,C 180,E1 -5827.665,E2 -5827.665} C_VEL
LIN {X 0,Y 503.563,Z 280.119,A -85,B 0,C 180,E1 -5830.43,E2 -5830.43} C_VEL
LIN {X 0,Y 503.084,Z 296.506,A -85,B 0,C 180,E1 -5833.358,E2 -5833.358} C_VEL
LIN {X 0,Y 502.767,Z 312.843,A -85,B 0,C 180,E1 -5836.253,E2 -5836.253} C_VEL
LIN {X 0,Y 502.664,Z 320.449,A -85,B 0,C 180,E1 -5837.576,E2 -5837.576} C_VEL
LIN {X 0,Y 504.114,Z 333.715,A -85,B 0,C 180,E1 -5837.801,E2 -5837.801} C_VEL
LIN {X 0,Y 503.819,Z 398.024,A -85,B 0,C 180,E1 -5838.738,E2 -5838.738} C_VEL
LIN {X 0,Y 503.59,Z 407.767,A -85,B 0,C 180,E1 -5838.988,E2 -5838.988} C_VEL
LIN {X 0,Y 503.403,Z 419.399,A -85,B 0,C 180,E1 -5839.441,E2 -5839.441} C_VEL
LIN {X 0,Y 503.163,Z 430.081,A -85,B 0,C 180,E1 -5840.046,E2 -5840.046} C_VEL
LIN {X 0,Y 502.978,Z 438.439,A -85,B 0,C 180,E1 -5840.652,E2 -5840.652} C_VEL
LIN {X 0,Y 502.748,Z 446.347,A -85,B 0,C 180,E1 -5841.357,E2 -5841.357} C_VEL
LIN {X 0,Y 502.521,Z 453.741,A -85,B 0,C 180,E1 -5842.163,E2 -5842.163} C_VEL
LIN {X 0,Y 502.403,Z 461.252,A -85,B 0,C 180,E1 -5843.171,E2 -5843.171} C_VEL
LIN {X 0,Y 502.26,Z 468.107,A -85,B 0,C 180,E1 -5844.379,E2 -5844.379} C_VEL
LIN {X 0,Y 502.133,Z 473.308,A -85,B 0,C 180,E1 -5845.585,E2 -5845.585} C_VEL
LIN {X 0,Y 502.165,Z 475.972,A -85,B 0,C 180,E1 -5846.389,E2 -5846.389} C_VEL
LIN {X 0,Y 502.124,Z 478.889,A -85,B 0,C 180,E1 -5847.593,E2 -5847.593} C_VEL
LIN {X 0,Y 502.036,Z 480.145,A -85,B 0,C 180,E1 -5848.395,E2 -5848.395} C_VEL
LIN {X 0,Y 501.994,Z 480.926,A -85,B 0,C 180,E1 -5849.198,E2 -5849.198} C_VEL
LIN {X 0,Y 501.99,Z 481.22,A -85,B 0,C 180,E1 -5850,E2 -5850} C_VEL
LIN {X 0,Y 501.994,Z 480.92,A -85,B 0,C 180,E1 -5850.802,E2 -5850.802} C_VEL
LIN {X 0,Y 502.036,Z 480.134,A -85,B 0,C 180,E1 -5851.604,E2 -5851.604} C_VEL
LIN {X 0,Y 502.124,Z 478.873,A -85,B 0,C 180,E1 -5852.406,E2 -5852.406} C_VEL
LIN {X 0,Y 502.165,Z 475.948,A -85,B 0,C 180,E1 -5853.611,E2 -5853.611} C_VEL
LIN {X 0,Y 502.133,Z 473.28,A -85,B 0,C 180,E1 -5854.415,E2 -5854.415} C_VEL
LIN {X 0,Y 502.26,Z 468.068,A -85,B 0,C 180,E1 -5855.621,E2 -5855.621} C_VEL
LIN {X 0,Y 502.37,Z 462.34,A -85,B 0,C 180,E1 -5856.648,E2 -5856.648} C_VEL
LIN {X 0,Y 502.499,Z 455.401,A -85,B 0,C 180,E1 -5857.635,E2 -5857.635} C_VEL
LIN {X 0,Y 502.705,Z 447.323,A -85,B 0,C 180,E1 -5858.542,E2 -5858.542} C_VEL
LIN {X 0,Y 502.913,Z 439.614,A -85,B 0,C 180,E1 -5859.248,E2 -5859.248} C_VEL
LIN {X 0,Y 503.122,Z 431.519,A -85,B 0,C 180,E1 -5859.853,E2 -5859.853} C_VEL
LIN {X 0,Y 503.29,Z 423.131,A -85,B 0,C 180,E1 -5860.357,E2 -5860.357} C_VEL
LIN {X 0,Y 503.473,Z 414.57,A -85,B 0,C 180,E1 -5860.76,E2 -5860.76} C_VEL
LIN {X 0,Y 503.681,Z 404.364,A -85,B 0,C 180,E1 -5861.112,E2 -5861.112} C_VEL
LIN {X 0,Y 503.905,Z 391.877,A -85,B 0,C 180,E1 -5861.37,E2 -5861.37} C_VEL
LIN {X 0,Y 504.03,Z 331.738,A -85,B 0,C 180,E1 -5862.227,E2 -5862.227} C_VEL
LIN {X 0,Y 502.644,Z 320.136,A -85,B 0,C 180,E1 -5862.438,E2 -5862.438} C_VEL
LIN {X 0,Y 502.898,Z 304.193,A -85,B 0,C 180,E1 -5865.236,E2 -5865.236} C_VEL
LIN {X 0,Y 503.344,Z 286.083,A -85,B 0,C 180,E1 -5868.44,E2 -5868.44} C_VEL
LIN {X 0,Y 503.78,Z 269.135,A -85,B 0,C 180,E1 -5871.481,E2 -5871.481} C_VEL
LIN {X 0,Y 503.756,Z 263.34,A -85,B 0,C 180,E1 -5872.539,E2 -5872.539} C_VEL
LIN {X 0,Y 502.822,Z 257.666,A -85,B 0,C 180,E1 -5873.639,E2 -5873.639} C_VEL
LIN {X 0,Y 502.87,Z 257.656,A -85,B 0,C 180,E1 -5876.566,E2 -5876.566} C_VEL
LIN {X 0,Y 502.827,Z 257.665,A -85,B 0,C 180,E1 -5879.287,E2 -5879.287} C_VEL
LIN {X 0,Y 502.787,Z 257.662,A -85,B 0,C 180,E1 -5882.084,E2 -5882.084} C_VEL
LIN {X 0,Y 502.8,Z 257.667,A -85,B 0,C 180,E1 -5884.966,E2 -5884.966} C_VEL
LIN {X 0,Y 502.797,Z 257.664,A -85,B 0,C 180,E1 -5887.953,E2 -5887.953} C_VEL
LIN {X 0,Y 502.825,Z 257.663,A -85,B 0,C 180,E1 -5891.065,E2 -5891.065} C_VEL
LIN {X 0,Y 502.791,Z 257.661,A -85,B 0,C 180,E1 -5894.529,E2 -5894.529} C_VEL
LIN {X 0,Y 502.801,Z 257.666,A -85,B 0,C 180,E1 -5897.86,E2 -5897.86} C_VEL
LIN {X 0,Y 502.8,Z 257.662,A -85,B 0,C 180,E1 -5901.022,E2 -5901.022} C_VEL
LIN {X 0,Y 502.781,Z 257.663,A -85,B 0,C 180,E1 -5904.168,E2 -5904.168} C_VEL
LIN {X 0,Y 502.837,Z 257.658,A -85,B 0,C 180,E1 -5906.993,E2 -5906.993} C_VEL
LIN {X 0,Y 502.82,Z 257.663,A -85,B 0,C 180,E1 -5910.064,E2 -5910.064} C_VEL
LIN {X 0,Y 502.851,Z 257.659,A -85,B 0,C 180,E1 -5913.442,E2 -5913.442} C_VEL
LIN {X 0,Y 502.78,Z 257.668,A -85,B 0,C 180,E1 -5916.084,E2 -5916.084} C_VEL
LIN {X 0,Y 502.787,Z 257.66,A -85,B 0,C 180,E1 -5918.687,E2 -5918.687} C_VEL
LIN {X 0,Y 502.828,Z 257.659,A -85,B 0,C 180,E1 -5921.246,E2 -5921.246} C_VEL
LIN {X 0,Y 502.854,Z 257.653,A -85,B 0,C 180,E1 -5924.598,E2 -5924.598} C_VEL
LIN {X 0,Y 502.881,Z 257.654,A -85,B 0,C 180,E1 -5928.037,E2 -5928.037} C_VEL
LIN {X 0,Y 502.872,Z 257.651,A -85,B 0,C 180,E1 -5931.154,E2 -5931.154} C_VEL
LIN {X 0,Y 502.913,Z 257.648,A -85,B 0,C 180,E1 -5933.579,E2 -5933.579} C_VEL
LIN {X 0,Y 502.865,Z 257.652,A -85,B 0,C 180,E1 -5936.793,E2 -5936.793} C_VEL
LIN {X 0,Y 502.896,Z 257.65,A -85,B 0,C 180,E1 -5938.396,E2 -5938.396} C_VEL
LIN {X 0,Y 502.99,Z 257.636,A -85,B 0,C 180,E1 -5940.798,E2 -5940.798} C_VEL
LIN {X 0,Y 503.019,Z 257.638,A -85,B 0,C 180,E1 -5942.4,E2 -5942.4} C_VEL
LIN {X 0,Y 502.921,Z 257.643,A -85,B 0,C 180,E1 -5945.611,E2 -5945.611} C_VEL
LIN {X 0,Y 502.865,Z 257.653,A -85,B 0,C 180,E1 -5948.841,E2 -5948.841} C_VEL
LIN {X 0,Y 502.841,Z 257.661,A -85,B 0,C 180,E1 -5952.099,E2 -5952.099} C_VEL
LIN {X 0,Y 502.842,Z 257.654,A -85,B 0,C 180,E1 -5955.397,E2 -5955.397} C_VEL
LIN {X 0,Y 502.817,Z 257.662,A -85,B 0,C 180,E1 -5958.749,E2 -5958.749} C_VEL
LIN {X 0,Y 502.773,Z 257.664,A -85,B 0,C 180,E1 -5961.308,E2 -5961.308} C_VEL
LIN {X 0,Y 502.773,Z 257.667,A -85,B 0,C 180,E1 -5963.911,E2 -5963.911} C_VEL
LIN {X 0,Y 502.851,Z 257.663,A -85,B 0,C 180,E1 -5966.563,E2 -5966.563} C_VEL
LIN {X 0,Y 502.81,Z 257.661,A -85,B 0,C 180,E1 -5969.285,E2 -5969.285} C_VEL
LIN {X 0,Y 502.768,Z 257.668,A -85,B 0,C 180,E1 -5972.081,E2 -5972.081} C_VEL
LIN {X 0,Y 502.789,Z 257.662,A -85,B 0,C 180,E1 -5974.962,E2 -5974.962} C_VEL
LIN {X 0,Y 502.773,Z 257.666,A -85,B 0,C 180,E1 -5977.951,E2 -5977.951} C_VEL
LIN {X 0,Y 502.802,Z 257.665,A -85,B 0,C 180,E1 -5981.062,E2 -5981.062} C_VEL
LIN {X 0,Y 502.758,Z 257.667,A -85,B 0,C 180,E1 -5983.373,E2 -5983.373} C_VEL
LIN {X 0,Y 502.764,Z 257.667,A -85,B 0,C 180,E1 -5985.658,E2 -5985.658} C_VEL
LIN {X 0,Y 502.812,Z 257.661,A -85,B 0,C 180,E1 -5987.862,E2 -5987.862} C_VEL
LIN {X 0,Y 502.794,Z 257.67,A -85,B 0,C 180,E1 -5991.023,E2 -5991.023} C_VEL
LIN {X 0,Y 502.758,Z 257.671,A -85,B 0,C 180,E1 -5994.164,E2 -5994.164} C_VEL
LIN {X 0,Y 502.759,Z 257.671,A -85,B 0,C 180,E1 -5995.985,E2 -5995.985} C_VEL
LIN {X 0,Y 502.423,Z 258.223,A -85,B 0,C 180,E1 -5996.428,E2 -5996.428} C_VEL
LIN {X 0,Y 501.341,Z 260.045,A -85,B 0,C 180,E1 -5996.945,E2 -5996.945} C_VEL
LIN {X 0,Y 496.304,Z 268.237,A -85,B 0,C 180,E1 -5998.568,E2 -5998.568} C_VEL
LIN {X 0,Y 495.628,Z 271.021,A -85,B 0,C 180,E1 -5999.17,E2 -5999.17} C_VEL
LIN {X 0,Y 495.648,Z 276.874,A -85,B 0,C 180,E1 -6000.455,E2 -6000.455} C_VEL
LIN {X 0,Y 497.303,Z 286.613,A -85,B 0,C 180,E1 -6000.642,E2 -6000.642} C_VEL
LIN {X 0,Y 496.933,Z 352.762,A -85,B 0,C 180,E1 -6001.619,E2 -6001.619} C_VEL
LIN {X 0,Y 496.806,Z 362.83,A -85,B 0,C 180,E1 -6001.885,E2 -6001.885} C_VEL
LIN {X 0,Y 496.677,Z 374.089,A -85,B 0,C 180,E1 -6002.335,E2 -6002.335} C_VEL
LIN {X 0,Y 496.423,Z 384.711,A -85,B 0,C 180,E1 -6002.948,E2 -6002.948} C_VEL
LIN {X 0,Y 496.232,Z 392.337,A -85,B 0,C 180,E1 -6003.505,E2 -6003.505} C_VEL
LIN {X 0,Y 495.965,Z 399.795,A -85,B 0,C 180,E1 -6004.168,E2 -6004.168} C_VEL
LIN {X 0,Y 495.773,Z 406.029,A -85,B 0,C 180,E1 -6004.832,E2 -6004.832} C_VEL
LIN {X 0,Y 495.605,Z 412.867,A -85,B 0,C 180,E1 -6005.717,E2 -6005.717} C_VEL
LIN {X 0,Y 495.432,Z 418.443,A -85,B 0,C 180,E1 -6006.597,E2 -6006.597} C_VEL
LIN {X 0,Y 495.266,Z 424.024,A -85,B 0,C 180,E1 -6007.692,E2 -6007.692} C_VEL
LIN {X 0,Y 495.159,Z 428.324,A -85,B 0,C 180,E1 -6008.781,E2 -6008.781} C_VEL
LIN {X 0,Y 495.078,Z 431.994,A -85,B 0,C 180,E1 -6010.081,E2 -6010.081} C_VEL
LIN {X 0,Y 494.99,Z 433.669,A -85,B 0,C 180,E1 -6010.94,E2 -6010.94} C_VEL
LIN {X 0,Y 494.974,Z 434.941,A -85,B 0,C 180,E1 -6012.033,E2 -6012.033} C_VEL
LIN {X 0,Y 494.982,Z 435.163,A -85,B 0,C 180,E1 -6013.503,E2 -6013.503} C_VEL
LIN {X 0,Y 494.999,Z 434.001,A -85,B 0,C 180,E1 -6014.88,E2 -6014.88} C_VEL
LIN {X 0,Y 495.051,Z 431.916,A -85,B 0,C 180,E1 -6016.034,E2 -6016.034} C_VEL
LIN {X 0,Y 495.155,Z 428.346,A -85,B 0,C 180,E1 -6017.291,E2 -6017.291} C_VEL
LIN {X 0,Y 495.235,Z 424.571,A -85,B 0,C 180,E1 -6018.269,E2 -6018.269} C_VEL
LIN {X 0,Y 495.401,Z 419.061,A -85,B 0,C 180,E1 -6019.373,E2 -6019.373} C_VEL
LIN {X 0,Y 495.504,Z 413.974,A -85,B 0,C 180,E1 -6020.201,E2 -6020.201} C_VEL
LIN {X 0,Y 495.677,Z 407.829,A -85,B 0,C 180,E1 -6021.027,E2 -6021.027} C_VEL
LIN {X 0,Y 495.962,Z 401.344,A -85,B 0,C 180,E1 -6021.751,E2 -6021.751} C_VEL
LIN {X 0,Y 496.127,Z 394.287,A -85,B 0,C 180,E1 -6022.41,E2 -6022.41} C_VEL
LIN {X 0,Y 496.343,Z 386.817,A -85,B 0,C 180,E1 -6022.985,E2 -6022.985} C_VEL
LIN {X 0,Y 496.511,Z 378.615,A -85,B 0,C 180,E1 -6023.498,E2 -6023.498} C_VEL
LIN {X 0,Y 496.667,Z 370.3,A -85,B 0,C 180,E1 -6023.908,E2 -6023.908} C_VEL
LIN {X 0,Y 496.815,Z 361.301,A -85,B 0,C 180,E1 -6024.241,E2 -6024.241} C_VEL
LIN {X 0,Y 496.916,Z 352.207,A -85,B 0,C 180,E1 -6024.471,E2 -6024.471} C_VEL
LIN {X 0,Y 497.146,Z 285.797,A -85,B 0,C 180,E1 -6025.452,E2 -6025.452} C_VEL
LIN {X 0,Y 495.688,Z 276.841,A -85,B 0,C 180,E1 -6025.63,E2 -6025.63} C_VEL
LIN {X 0,Y 495.757,Z 263.237,A -85,B 0,C 180,E1 -6028.782,E2 -6028.782} C_VEL
LIN {X 0,Y 495.784,Z 258.54,A -85,B 0,C 180,E1 -6029.899,E2 -6029.899} C_VEL
LIN {X 0,Y 495.968,Z 258.519,A -85,B 0,C 180,E1 -6030.812,E2 -6030.812} C_VEL
LIN {X 0,Y 495.81,Z 258.541,A -85,B 0,C 180,E1 -6033.251,E2 -6033.251} C_VEL
LIN {X 0,Y 495.822,Z 258.531,A -85,B 0,C 180,E1 -6036.511,E2 -6036.511} C_VEL
LIN {X 0,Y 495.803,Z 258.537,A -85,B 0,C 180,E1 -6038.971,E2 -6038.971} C_VEL
LIN {X 0,Y 495.792,Z 258.535,A -85,B 0,C 180,E1 -6042.037,E2 -6042.037} C_VEL
LIN {X 0,Y 495.786,Z 258.543,A -85,B 0,C 180,E1 -6045.453,E2 -6045.453} C_VEL
LIN {X 0,Y 495.771,Z 258.537,A -85,B 0,C 180,E1 -6048.249,E2 -6048.249} C_VEL
LIN {X 0,Y 495.738,Z 258.542,A -85,B 0,C 180,E1 -6050.758,E2 -6050.758} C_VEL
LIN {X 0,Y 495.704,Z 258.554,A -85,B 0,C 180,E1 -6053.39,E2 -6053.39} C_VEL
LIN {X 0,Y 495.74,Z 258.541,A -85,B 0,C 180,E1 -6056.74,E2 -6056.74} C_VEL
LIN {X 0,Y 495.73,Z 258.547,A -85,B 0,C 180,E1 -6059.749,E2 -6059.749} C_VEL
LIN {X 0,Y 495.736,Z 258.541,A -85,B 0,C 180,E1 -6062.597,E2 -6062.597} C_VEL
LIN {X 0,Y 495.715,Z 258.553,A -85,B 0,C 180,E1 -6065.541,E2 -6065.541} C_VEL
LIN {X 0,Y 495.729,Z 258.543,A -85,B 0,C 180,E1 -6068.77,E2 -6068.77} C_VEL
LIN {X 0,Y 495.719,Z 258.55,A -85,B 0,C 180,E1 -6071.785,E2 -6071.785} C_VEL
LIN {X 0,Y 495.713,Z 258.547,A -85,B 0,C 180,E1 -6075.144,E2 -6075.144} C_VEL
LIN {X 0,Y 495.734,Z 258.543,A -85,B 0,C 180,E1 -6078.222,E2 -6078.222} C_VEL
LIN {X 0,Y 495.729,Z 258.547,A -85,B 0,C 180,E1 -6081.411,E2 -6081.411} C_VEL
LIN {X 0,Y 495.729,Z 258.543,A -85,B 0,C 180,E1 -6084.465,E2 -6084.465} C_VEL
LIN {X 0,Y 495.751,Z 258.544,A -85,B 0,C 180,E1 -6087.409,E2 -6087.409} C_VEL
LIN {X 0,Y 495.749,Z 258.542,A -85,B 0,C 180,E1 -6090.257,E2 -6090.257} C_VEL
LIN {X 0,Y 495.747,Z 258.543,A -85,B 0,C 180,E1 -6093.269,E2 -6093.269} C_VEL
LIN {X 0,Y 495.732,Z 258.543,A -85,B 0,C 180,E1 -6096.616,E2 -6096.616} C_VEL
LIN {X 0,Y 495.771,Z 258.54,A -85,B 0,C 180,E1 -6099.327,E2 -6099.327} C_VEL
LIN {X 0,Y 495.773,Z 258.545,A -85,B 0,C 180,E1 -6101.832,E2 -6101.832} C_VEL
LIN {X 0,Y 495.764,Z 258.563,A -85,B 0,C 180,E1 -6103.162,E2 -6103.162} C_VEL
LIN {X 0,Y 495.72,Z 268.944,A -85,B 0,C 180,E1 -6105.638,E2 -6105.638} C_VEL
LIN {X 0,Y 495.598,Z 276.756,A -85,B 0,C 180,E1 -6107.499,E2 -6107.499} C_VEL
LIN {X 0,Y 497.171,Z 287.334,A -85,B 0,C 180,E1 -6107.714,E2 -6107.714} C_VEL
LIN {X 0,Y 496.756,Z 353.418,A -85,B 0,C 180,E1 -6108.76,E2 -6108.76} C_VEL
LIN {X 0,Y 496.631,Z 363.345,A -85,B 0,C 180,E1 -6109.041,E2 -6109.041} C_VEL
LIN {X 0,Y 496.435,Z 372.225,A -85,B 0,C 180,E1 -6109.398,E2 -6109.398} C_VEL
LIN {X 0,Y 496.298,Z 380.067,A -85,B 0,C 180,E1 -6109.807,E2 -6109.807} C_VEL
LIN {X 0,Y 496.134,Z 389.363,A -85,B 0,C 180,E1 -6110.422,E2 -6110.422} C_VEL
LIN {X 0,Y 495.895,Z 399.101,A -85,B 0,C 180,E1 -6111.24,E2 -6111.24} C_VEL
LIN {X 0,Y 495.686,Z 406.718,A -85,B 0,C 180,E1 -6112.057,E2 -6112.057} C_VEL
LIN {X 0,Y 495.495,Z 413.242,A -85,B 0,C 180,E1 -6112.91,E2 -6112.91} C_VEL
LIN {X 0,Y 495.506,Z 418.221,A -85,B 0,C 180,E1 -6113.692,E2 -6113.692} C_VEL
LIN {X 0,Y 495.204,Z 423.516,A -85,B 0,C 180,E1 -6114.71,E2 -6114.71} C_VEL
LIN {X 0,Y 495.251,Z 426.929,A -85,B 0,C 180,E1 -6115.526,E2 -6115.526} C_VEL
LIN {X 0,Y 495.149,Z 430.849,A -85,B 0,C 180,E1 -6116.748,E2 -6116.748} C_VEL
LIN {X 0,Y 495.07,Z 432.714,A -85,B 0,C 180,E1 -6117.562,E2 -6117.562} C_VEL
LIN {X 0,Y 494.965,Z 434.06,A -85,B 0,C 180,E1 -6118.375,E2 -6118.375} C_VEL
LIN {X 0,Y 494.92,Z 434.909,A -85,B 0,C 180,E1 -6119.189,E2 -6119.189} C_VEL
LIN {X 0,Y 494.914,Z 435.233,A -85,B 0,C 180,E1 -6120.003,E2 -6120.003} C_VEL
LIN {X 0,Y 494.921,Z 434.976,A -85,B 0,C 180,E1 -6120.816,E2 -6120.816} C_VEL
LIN {X 0,Y 494.966,Z 434.222,A -85,B 0,C 180,E1 -6121.63,E2 -6121.63} C_VEL
LIN {X 0,Y 495.073,Z 432.969,A -85,B 0,C 180,E1 -6122.443,E2 -6122.443} C_VEL
LIN {X 0,Y 495.172,Z 430.078,A -85,B 0,C 180,E1 -6123.664,E2 -6123.664} C_VEL
LIN {X 0,Y 495.235,Z 425.903,A -85,B 0,C 180,E1 -6124.887,E2 -6124.887} C_VEL
LIN {X 0,Y 495.371,Z 421.186,A -85,B 0,C 180,E1 -6125.906,E2 -6125.906} C_VEL
LIN {X 0,Y 495.487,Z 414.95,A -85,B 0,C 180,E1 -6126.961,E2 -6126.961} C_VEL
LIN {X 0,Y 495.635,Z 409.295,A -85,B 0,C 180,E1 -6127.744,E2 -6127.744} C_VEL
LIN {X 0,Y 495.836,Z 402.15,A -85,B 0,C 180,E1 -6128.561,E2 -6128.561} C_VEL
LIN {X 0,Y 496.062,Z 393.346,A -85,B 0,C 180,E1 -6129.379,E2 -6129.379} C_VEL
LIN {X 0,Y 496.327,Z 383.44,A -85,B 0,C 180,E1 -6130.094,E2 -6130.094} C_VEL
LIN {X 0,Y 496.488,Z 373.09,A -85,B 0,C 180,E1 -6130.658,E2 -6130.658} C_VEL
LIN {X 0,Y 496.614,Z 363.624,A -85,B 0,C 180,E1 -6131.042,E2 -6131.042} C_VEL
LIN {X 0,Y 496.775,Z 352.583,A -85,B 0,C 180,E1 -6131.348,E2 -6131.348} C_VEL
LIN {X 0,Y 497.142,Z 285.763,A -85,B 0,C 180,E1 -6132.416,E2 -6132.416} C_VEL
LIN {X 0,Y 495.676,Z 277.494,A -85,B 0,C 180,E1 -6132.604,E2 -6132.604} C_VEL
LIN {X 0,Y 495.79,Z 264.435,A -85,B 0,C 180,E1 -6135.627,E2 -6135.627} C_VEL
LIN {X 0,Y 495.831,Z 258.538,A -85,B 0,C 180,E1 -6137,E2 -6137} C_VEL
LIN {X 0,Y 495.777,Z 258.546,A -85,B 0,C 180,E1 -6139.892,E2 -6139.892} C_VEL
LIN {X 0,Y 495.767,Z 258.541,A -85,B 0,C 180,E1 -6142.862,E2 -6142.862} C_VEL
LIN {X 0,Y 495.732,Z 258.55,A -85,B 0,C 180,E1 -6146.073,E2 -6146.073} C_VEL
LIN {X 0,Y 495.751,Z 258.544,A -85,B 0,C 180,E1 -6148.818,E2 -6148.818} C_VEL
LIN {X 0,Y 495.762,Z 258.541,A -85,B 0,C 180,E1 -6151.726,E2 -6151.726} C_VEL
LIN {X 0,Y 495.769,Z 258.544,A -85,B 0,C 180,E1 -6154.693,E2 -6154.693} C_VEL
LIN {X 0,Y 495.729,Z 258.544,A -85,B 0,C 180,E1 -6157.563,E2 -6157.563} C_VEL
LIN {X 0,Y 495.753,Z 258.543,A -85,B 0,C 180,E1 -6160.046,E2 -6160.046} C_VEL
LIN {X 0,Y 495.725,Z 258.547,A -85,B 0,C 180,E1 -6162.885,E2 -6162.885} C_VEL
LIN {X 0,Y 495.732,Z 258.544,A -85,B 0,C 180,E1 -6165.999,E2 -6165.999} C_VEL
LIN {X 0,Y 495.745,Z 258.548,A -85,B 0,C 180,E1 -6168.71,E2 -6168.71} C_VEL
LIN {X 0,Y 495.754,Z 258.54,A -85,B 0,C 180,E1 -6171.408,E2 -6171.408} C_VEL
LIN {X 0,Y 495.751,Z 258.545,A -85,B 0,C 180,E1 -6174.462,E2 -6174.462} C_VEL
LIN {X 0,Y 495.758,Z 258.541,A -85,B 0,C 180,E1 -6177.405,E2 -6177.405} C_VEL
LIN {X 0,Y 495.772,Z 258.541,A -85,B 0,C 180,E1 -6180.254,E2 -6180.254} C_VEL
LIN {X 0,Y 495.83,Z 258.534,A -85,B 0,C 180,E1 -6183.251,E2 -6183.251} C_VEL
LIN {X 0,Y 495.799,Z 258.623,A -85,B 0,C 180,E1 -6186.2,E2 -6186.2} C_VEL
LIN {X 0,Y 496.909,Z 265.64,A -85,B 0,C 180,E1 -6187.55,E2 -6187.55} C_VEL
LIN {X 0,Y 496.538,Z 280.937,A -85,B 0,C 180,E1 -6190.357,E2 -6190.357} C_VEL
LIN {X 0,Y 496.028,Z 297.335,A -85,B 0,C 180,E1 -6193.327,E2 -6193.327} C_VEL
LIN {X 0,Y 495.714,Z 313.678,A -85,B 0,C 180,E1 -6196.262,E2 -6196.262} C_VEL
LIN {X 0,Y 495.614,Z 319.94,A -85,B 0,C 180,E1 -6197.381,E2 -6197.381} C_VEL
LIN {X 0,Y 497.16,Z 334.33,A -85,B 0,C 180,E1 -6197.643,E2 -6197.643} C_VEL
LIN {X 0,Y 496.868,Z 397.572,A -85,B 0,C 180,E1 -6198.578,E2 -6198.578} C_VEL
LIN {X 0,Y 496.636,Z 407.366,A -85,B 0,C 180,E1 -6198.831,E2 -6198.831} C_VEL
LIN {X 0,Y 496.414,Z 419.034,A -85,B 0,C 180,E1 -6199.291,E2 -6199.291} C_VEL
LIN {X 0,Y 496.142,Z 429.733,A -85,B 0,C 180,E1 -6199.904,E2 -6199.904} C_VEL
LIN {X 0,Y 495.965,Z 438.102,A -85,B 0,C 180,E1 -6200.518,E2 -6200.518} C_VEL
LIN {X 0,Y 495.706,Z 446.015,A -85,B 0,C 180,E1 -6201.233,E2 -6201.233} C_VEL
LIN {X 0,Y 495.453,Z 453.41,A -85,B 0,C 180,E1 -6202.05,E2 -6202.05} C_VEL
LIN {X 0,Y 495.336,Z 460.923,A -85,B 0,C 180,E1 -6203.073,E2 -6203.073} C_VEL
LIN {X 0,Y 495.19,Z 467.78,A -85,B 0,C 180,E1 -6204.298,E2 -6204.298} C_VEL
LIN {X 0,Y 495.038,Z 472.98,A -85,B 0,C 180,E1 -6205.521,E2 -6205.521} C_VEL
LIN {X 0,Y 495.086,Z 475.646,A -85,B 0,C 180,E1 -6206.337,E2 -6206.337} C_VEL
LIN {X 0,Y 495.028,Z 478.563,A -85,B 0,C 180,E1 -6207.559,E2 -6207.559} C_VEL
LIN {X 0,Y 494.963,Z 479.82,A -85,B 0,C 180,E1 -6208.373,E2 -6208.373} C_VEL
LIN {X 0,Y 494.914,Z 480.601,A -85,B 0,C 180,E1 -6209.186,E2 -6209.186} C_VEL
LIN {X 0,Y 494.907,Z 480.894,A -85,B 0,C 180,E1 -6210,E2 -6210} C_VEL
LIN {X 0,Y 494.914,Z 480.593,A -85,B 0,C 180,E1 -6210.813,E2 -6210.813} C_VEL
LIN {X 0,Y 494.963,Z 479.806,A -85,B 0,C 180,E1 -6211.627,E2 -6211.627} C_VEL
LIN {X 0,Y 495.028,Z 478.544,A -85,B 0,C 180,E1 -6212.441,E2 -6212.441} C_VEL
LIN {X 0,Y 495.086,Z 475.618,A -85,B 0,C 180,E1 -6213.662,E2 -6213.662} C_VEL
LIN {X 0,Y 495.038,Z 472.947,A -85,B 0,C 180,E1 -6214.478,E2 -6214.478} C_VEL
LIN {X 0,Y 495.19,Z 467.733,A -85,B 0,C 180,E1 -6215.701,E2 -6215.701} C_VEL
LIN {X 0,Y 495.341,Z 461.133,A -85,B 0,C 180,E1 -6216.886,E2 -6216.886} C_VEL
LIN {X 0,Y 495.452,Z 453.354,A -85,B 0,C 180,E1 -6217.95,E2 -6217.95} C_VEL
LIN {X 0,Y 495.705,Z 445.962,A -85,B 0,C 180,E1 -6218.767,E2 -6218.767} C_VEL
LIN {X 0,Y 495.95,Z 438.05,A -85,B 0,C 180,E1 -6219.482,E2 -6219.482} C_VEL
LIN {X 0,Y 496.141,Z 429.691,A -85,B 0,C 180,E1 -6220.096,E2 -6220.096} C_VEL
LIN {X 0,Y 496.395,Z 419.022,A -85,B 0,C 180,E1 -6220.709,E2 -6220.709} C_VEL
LIN {X 0,Y 496.633,Z 407.418,A -85,B 0,C 180,E1 -6221.168,E2 -6221.168} C_VEL
LIN {X 0,Y 496.848,Z 397.715,A -85,B 0,C 180,E1 -6221.422,E2 -6221.422} C_VEL
LIN {X 0,Y 497.138,Z 332.628,A -85,B 0,C 180,E1 -6222.385,E2 -6222.385} C_VEL
LIN {X 0,Y 495.583,Z 319.758,A -85,B 0,C 180,E1 -6222.628,E2 -6222.628} C_VEL
LIN {X 0,Y 495.935,Z 302.954,A -85,B 0,C 180,E1 -6225.62,E2 -6225.62} C_VEL
LIN {X 0,Y 496.338,Z 286.153,A -85,B 0,C 180,E1 -6228.643,E2 -6228.643} C_VEL
LIN {X 0,Y 496.8,Z 268.84,A -85,B 0,C 180,E1 -6231.799,E2 -6231.799} C_VEL
LIN {X 0,Y 496.683,Z 263.75,A -85,B 0,C 180,E1 -6232.747,E2 -6232.747} C_VEL
LIN {X 0,Y 495.763,Z 258.545,A -85,B 0,C 180,E1 -6233.774,E2 -6233.774} C_VEL
LIN {X 0,Y 495.817,Z 258.539,A -85,B 0,C 180,E1 -6236.974,E2 -6236.974} C_VEL
LIN {X 0,Y 495.769,Z 258.538,A -85,B 0,C 180,E1 -6240.146,E2 -6240.146} C_VEL
LIN {X 0,Y 495.757,Z 258.544,A -85,B 0,C 180,E1 -6243.236,E2 -6243.236} C_VEL
LIN {X 0,Y 495.724,Z 258.542,A -85,B 0,C 180,E1 -6246.088,E2 -6246.088} C_VEL
LIN {X 0,Y 495.768,Z 258.539,A -85,B 0,C 180,E1 -6248.767,E2 -6248.767} C_VEL
LIN {X 0,Y 495.762,Z 258.543,A -85,B 0,C 180,E1 -6251.78,E2 -6251.78} C_VEL
LIN {X 0,Y 495.743,Z 258.543,A -85,B 0,C 180,E1 -6255.14,E2 -6255.14} C_VEL
LIN {X 0,Y 495.757,Z 258.54,A -85,B 0,C 180,E1 -6258.217,E2 -6258.217} C_VEL
LIN {X 0,Y 495.752,Z 258.544,A -85,B 0,C 180,E1 -6261.407,E2 -6261.407} C_VEL
LIN {X 0,Y 495.753,Z 258.537,A -85,B 0,C 180,E1 -6264.461,E2 -6264.461} C_VEL
LIN {X 0,Y 495.772,Z 258.542,A -85,B 0,C 180,E1 -6267.404,E2 -6267.404} C_VEL
LIN {X 0,Y 495.768,Z 258.539,A -85,B 0,C 180,E1 -6270.252,E2 -6270.252} C_VEL
LIN {X 0,Y 495.781,Z 258.537,A -85,B 0,C 180,E1 -6273.261,E2 -6273.261} C_VEL
LIN {X 0,Y 495.729,Z 258.55,A -85,B 0,C 180,E1 -6275.722,E2 -6275.722} C_VEL
LIN {X 0,Y 495.747,Z 258.538,A -85,B 0,C 180,E1 -6278.369,E2 -6278.369} C_VEL
LIN {X 0,Y 495.784,Z 258.535,A -85,B 0,C 180,E1 -6280.97,E2 -6280.97} C_VEL
LIN {X 0,Y 495.829,Z 258.529,A -85,B 0,C 180,E1 -6284.547,E2 -6284.547} C_VEL
LIN {X 0,Y 495.833,Z 258.533,A -85,B 0,C 180,E1 -6287.963,E2 -6287.963} C_VEL
LIN {X 0,Y 495.841,Z 258.526,A -85,B 0,C 180,E1 -6291.028,E2 -6291.028} C_VEL
LIN {X 0,Y 495.866,Z 258.525,A -85,B 0,C 180,E1 -6293.487,E2 -6293.487} C_VEL
LIN {X 0,Y 495.722,Z 258.546,A -85,B 0,C 180,E1 -6295.933,E2 -6295.933} C_VEL
LIN {X 0,Y 495.987,Z 258.511,A -85,B 0,C 180,E1 -6297.561,E2 -6297.561} C_VEL
LIN {X 0,Y 495.942,Z 258.514,A -85,B 0,C 180,E1 -6300.809,E2 -6300.809} C_VEL
LIN {X 0,Y 495.986,Z 258.514,A -85,B 0,C 180,E1 -6302.434,E2 -6302.434} C_VEL
LIN {X 0,Y 495.876,Z 258.522,A -85,B 0,C 180,E1 -6305.691,E2 -6305.691} C_VEL
LIN {X 0,Y 495.834,Z 258.529,A -85,B 0,C 180,E1 -6308.967,E2 -6308.967} C_VEL
LIN {X 0,Y 495.823,Z 258.534,A -85,B 0,C 180,E1 -6312.032,E2 -6312.032} C_VEL
LIN {X 0,Y 495.817,Z 258.529,A -85,B 0,C 180,E1 -6315.448,E2 -6315.448} C_VEL
LIN {X 0,Y 495.77,Z 258.545,A -85,B 0,C 180,E1 -6318.234,E2 -6318.234} C_VEL
LIN {X 0,Y 495.764,Z 258.541,A -85,B 0,C 180,E1 -6320.753,E2 -6320.753} C_VEL
LIN {X 0,Y 495.736,Z 258.541,A -85,B 0,C 180,E1 -6323.384,E2 -6323.384} C_VEL
LIN {X 0,Y 495.778,Z 258.539,A -85,B 0,C 180,E1 -6326.065,E2 -6326.065} C_VEL
LIN {X 0,Y 495.758,Z 258.543,A -85,B 0,C 180,E1 -6328.812,E2 -6328.812} C_VEL
LIN {X 0,Y 495.739,Z 258.54,A -85,B 0,C 180,E1 -6331.722,E2 -6331.722} C_VEL
LIN {X 0,Y 495.756,Z 258.542,A -85,B 0,C 180,E1 -6334.692,E2 -6334.692} C_VEL
LIN {X 0,Y 495.71,Z 258.545,A -85,B 0,C 180,E1 -6337.558,E2 -6337.558} C_VEL
LIN {X 0,Y 495.748,Z 258.545,A -85,B 0,C 180,E1 -6340.697,E2 -6340.697} C_VEL
LIN {X 0,Y 495.71,Z 258.544,A -85,B 0,C 180,E1 -6343.692,E2 -6343.692} C_VEL
LIN {X 0,Y 495.709,Z 258.55,A -85,B 0,C 180,E1 -6346.302,E2 -6346.302} C_VEL
LIN {X 0,Y 495.755,Z 258.543,A -85,B 0,C 180,E1 -6349.299,E2 -6349.299} C_VEL
LIN {X 0,Y 495.736,Z 258.546,A -85,B 0,C 180,E1 -6351.407,E2 -6351.407} C_VEL
LIN {X 0,Y 495.731,Z 258.549,A -85,B 0,C 180,E1 -6354.461,E2 -6354.461} C_VEL
LIN {X 0,Y 495.679,Z 258.664,A -85,B 0,C 180,E1 -6356.43,E2 -6356.43} C_VEL
LIN {X 0,Y 495.636,Z 269.5,A -85,B 0,C 180,E1 -6358.831,E2 -6358.831} C_VEL
LIN {X 0,Y 495.628,Z 271.021,A -85,B 0,C 180,E1 -6359.17,E2 -6359.17} C_VEL
LIN {X 0,Y 495.388,Z 273.239,A -85,B 0,C 180,E1 -6359.533,E2 -6359.533} C_VEL
LIN {X 0,Y 494.389,Z 277.696,A -85,B 0,C 180,E1 -6359.954,E2 -6359.954} C_VEL
LIN {X 0,Y 493.032,Z 282.892,A -85,B 0,C 180,E1 -6360.242,E2 -6360.242} C_VEL
LIN {X 0,Y 491.205,Z 290.728,A -85,B 0,C 180,E1 -6360.488,E2 -6360.488} C_VEL
